# B&R Automation Studio project SuperTrak_Core
Automation Studio 4.7.4.67 SP; technology packages: mapp 5.11.1, mappView 5.11.2

## Configuration Simulation

CPU PC_any, AutomationRuntime B4.62, Build 4.1.2, Safety 0.0, Vc not defined

### Task classes (Cpu.sw)
```
Cyclic#1 (cycle 800 us, tolerance 0 us):
  ST_MainSim <- Source.ST_Core.ST_Main.prg
  ST_Logic <- Source.ST_Core.ST_Logic.prg
Cyclic#2 (cycle 800 us, tolerance 0 us):
  MainCtrl <- Source.Main.MainCtrl.prg
Cyclic#3 (cycle 50000 us):
  Alarms <- Source.Main.Alarms.prg
Cyclic#8 (cycle 800 us, tolerance 0 us):
  ST_Visu <- Source.ST_Core.ST_Visu.prg
DataObjects: Acp10sys, McAcpSys
Binaries: udbdef, mvLoader, TCData, arsvcreg, ashwac, arconfig, asfw, ashwd, iomap, User, Role, sysconf, Config_1, Config, Config_2, OpcUaMap, Acp10map, acp10cfg, McProfGen, McAcpSim, McAcpDrv, Config_3
Libraries: AsGuard, operator, runtime, astime, DevDetect, AsUDP, AsETH, AsIOTime, AsARCfg, AsIecCon, AsBrStr, AsIODiag, standard, ArEventLog, sys_lib, AsTCP, FileIO, brsystem, AsMem, DataObj, SuperTrak, AsArProf, StCom, CoTrace, AsZip, asstring, AsEthIP, AsPciStr, AsBrMath, MpAlarmX, MpBase, MpServer, MpCom, AsArLog, NcGlobal, aspciext, aruser, powerlnk
```

### Hardware
```
5LS182.6-2 : 5LS182.6-2 v1.3.1.0  [SL -> PC.SL4]
PC : PC_any v1.1.0.0 (OrderNumber=PC)
  Connector IF3:
    InaPort = 11159
  ConfigurationID = SuperTrak_Core_Simulation
  VolatileGlobalPvSize = 131070
  SystemTick = 400
  TaskClassIdleTime = 400
  Cyclic1Duration = 800
  Cyclic1Tolerance = 0
  Cyclic1Stack = 65535
  Cyclic1Output = 1
  Cyclic2Duration = 800
  Cyclic2Tolerance = 0
  Cyclic2Stack = 65535
  Cyclic3Duration = 50000
  Cyclic8Duration = 800
  Cyclic8Tolerance = 0
  FileDevice1
  FileDeviceName1 = USER
  FileDevicePath1 = ../../../../Logical/ConfigFiles
  FtpUser1
  FtpUsername1 = br
  FtpUserPassword1 = QMhL/dtrmhlR40mhXiUTZRHGDCdjSPoAwBd7aMiCRQw=
  FtpUserSalt1 = /GvO8l4J
  FTPAccessRight1 = 0
  WebServerWebDir = C:\web\
  ActivateOpcUa = 1
  OpcUaInformationModels_PV_Version = 1
```

## Configuration Standard_PC_TS77_04

CPU 5PC900.TS77-04, AutomationRuntime C4.72, Build 4.1.2, Safety 1.10, Vc V4.33.0

### Task classes (Cpu.sw)
```
Cyclic#1 (cycle 800 us, tolerance 0 us):
  ST_Main <- Source.ST_Core.ST_Main.prg
  ST_Logic <- Source.ST_Core.ST_Logic.prg
Cyclic#2 (cycle 800 us, tolerance 0 us):
  MainCtrl <- Source.Main.MainCtrl.prg
Cyclic#3:
  Alarms <- Source.Main.Alarms.prg
Cyclic#4:
  ST_Visu <- Source.ST_Core.ST_Visu.prg
Binaries: udbdef, mvLoader, TCData, arsvcreg, arconfig, User, Config, ashwd, Config_1, sysconf, ashwac, Role, asfw, iomap
Libraries: AsBrMath, AsGuard, operator, runtime, astime, DevDetect, AsUDP, AsETH, AsIOTime, AsARCfg, AsIecCon, AsBrStr, AsIODiag, standard, ArEventLog, sys_lib, AsTCP, FileIO, brsystem, AsMem, DataObj, SuperTrak, AsArProf, StCom, AsZip, asstring, AsEthIP, AsPciStr, MpBase, CoTrace, aruser, AsArLog, McBase, MpCom, MpAlarmX, MpServer, AsIOAcc
```

### Hardware
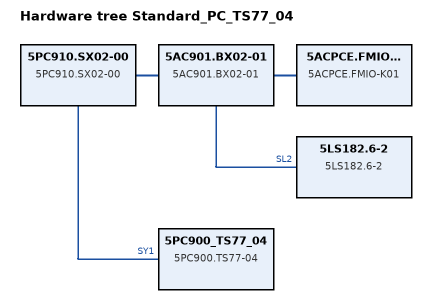
```
5AC901.BX02-01 : 5AC901.BX02-01 v1.1.1.0  [SY -> 5PC910.SX02-00.SY3]
5ACPCE.FMIO-K01 : 5ACPCE.FMIO-K01 v1.0.6.0  [SL -> 5AC901.BX02-01.SL1]
5LS182.6-2 : 5LS182.6-2 v1.4.0.0  [SL -> 5AC901.BX02-01.SL2]
  Connector IF1:
    CycleTime = 400
5PC900_TS77_04 : 5PC900.TS77-04 v2.0.1.0  [SY -> 5PC910.SX02-00.SY1]
  ConfigurationID = SuperTrak_Core_Standard_PC_TS77_04
  UserPartitionSize = 200
  RemMemDevice = PCI.2.LS182.SRAM
  RemMemSize = 500
  SystemTick = 400
  TaskClassIdleTime = 400
  Cyclic1Duration = 800
  Cyclic1Tolerance = 0
  Cyclic1Output = 1
  Cyclic2Duration = 800
  Cyclic2Tolerance = 0
  FileDevice1
  FileDeviceName1 = USER
  FileDevicePath1 = F:\SuperTrakCore
  EthernetDefaultGateway = 10.1.60.1
  ActivateDns = 1
  DnsDefaultDomain = br-automation.com
  DnsServer1 = 10.1.10.30
  FtpUser1
  FtpUsername1 = br
  FtpUserPassword1 = WcK/x6vgpRURITa0IoUtKo9v6R/fBL8dK5K21ruWyPI=
  FtpUserSalt1 = AV6KF4Bt
  FTPAccessRight1 = 0
  ActivateOpcUa = 1
  OpcUaInformationModels_PV_Version = 1
5PC910.SX02-00 : 5PC910.SX02-00 v2.0.2.0
  Connector IF1:
    AssignedOperatingSystem = ARemb
  Connector IF3:
    AssignedOperatingSystem = ARemb
    ActivateDevice = 1
    Mode = Manual
    InternetAddress = 10.1.60.55
    SubnetMask = 255.255.255.0
  Connector IF4:
    AssignedOperatingSystem = ARemb
    ActivateDevice = 1
    Mode = Manual
    InternetAddress = 10.11.10.12
    SubnetMask = 255.255.255.0
  Connector IF5:
    AssignedOperatingSystem = ARemb
  Connector IF6:
    AssignedOperatingSystem = ARemb
  Connector IF7:
    AssignedOperatingSystem = ARemb
  Connector IF8:
    AssignedOperatingSystem = ARemb
  Connector IF9:
    AssignedOperatingSystem = ARemb
```

## Configuration Standard_PC_TS77_1

CPU 5PC900.TS77-04, AutomationRuntime B4.45, Build 4.1.2, Vc V4.33.0, Safety 1.10

### Task classes (Cpu.sw)
```
Cyclic#1 (cycle 800 us, tolerance 0 us):
  ST_Main <- Source.ST_Core.ST_Main.prg
  ST_Logic <- Source.ST_Core.ST_Logic.prg
Cyclic#2 (cycle 800 us, tolerance 0 us):
  MainCtrl <- Source.Main.MainCtrl.prg
Cyclic#3:
  Alarms <- Source.Main.Alarms.prg
Cyclic#4:
  ST_Visu <- Source.ST_Core.ST_Visu.prg
Binaries: udbdef, mvLoader, TCData, arsvcreg, arconfig, User, Config, ashwd, Config_1, sysconf, ashwac, Role, asfw, iomap
Libraries: AsBrMath, AsGuard, operator, runtime, astime, DevDetect, AsUDP, AsETH, AsIOTime, AsARCfg, AsIecCon, AsBrStr, AsIODiag, standard, ArEventLog, sys_lib, AsTCP, FileIO, brsystem, AsMem, DataObj, SuperTrak, AsArProf, StCom, AsZip, asstring, AsEthIP, AsPciStr, MpBase, CoTrace, aruser, AsArLog, McBase, MpCom, MpAlarmX, MpServer
```

### Hardware
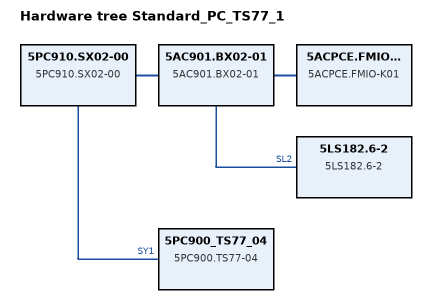
```
5AC901.BX02-01 : 5AC901.BX02-01 v1.1.1.0  [SY -> 5PC910.SX02-00.SY3]
5ACPCE.FMIO-K01 : 5ACPCE.FMIO-K01 v1.0.6.0  [SL -> 5AC901.BX02-01.SL1]
5LS182.6-2 : 5LS182.6-2 v1.3.1.0  [SL -> 5AC901.BX02-01.SL2]
  Connector IF1:
    CycleTime = 400
5PC900_TS77_04 : 5PC900.TS77-04 v2.0.0.0  [SY -> 5PC910.SX02-00.SY1]
  ConfigurationID = SuperTrak_Core_Standard_PC_TS77_04
  UserPartitionSize = 200
  RemMemDevice = PCI.2.LS182.SRAM
  RemMemSize = 500
  SystemTick = 400
  TaskClassIdleTime = 400
  Cyclic1Duration = 800
  Cyclic1Tolerance = 0
  Cyclic1Output = 1
  Cyclic2Duration = 800
  Cyclic2Tolerance = 0
  FileDevice1
  FileDeviceName1 = USER
  FileDevicePath1 = F:\SuperTrakCore
  FtpUser1
  FtpUsername1 = br
  FtpUserPassword1 = WcK/x6vgpRURITa0IoUtKo9v6R/fBL8dK5K21ruWyPI=
  FtpUserSalt1 = AV6KF4Bt
  FTPAccessRight1 = 0
  ActivateOpcUa = 1
  OpcUaInformationModels_PV_Version = 1
5PC910.SX02-00 : 5PC910.SX02-00 v2.0.1.0
  Connector IF1:
    AssignedOperatingSystem = ARemb
  Connector IF3:
    AssignedOperatingSystem = ARemb
    ActivateDevice = 1
    Mode = Manual
    InternetAddress = 10.11.10.50
    SubnetMask = 255.255.255.0
  Connector IF4:
    ActivateDevice = 1
    Mode = Manual
    InternetAddress = 10.1.10.11
    SubnetMask = 255.255.255.0
  Connector IF5:
    AssignedOperatingSystem = ARemb
  Connector IF6:
    AssignedOperatingSystem = ARemb
  Connector IF7:
    AssignedOperatingSystem = ARemb
  Connector IF8:
    AssignedOperatingSystem = ARemb
  Connector IF9:
    AssignedOperatingSystem = ARemb
```

### Config.mpalarmxcore - 5PC900_TS77_04/mappServices/Config.mpalarmxcore
```
Element gAlarmXCore (Type=mpalarmxcore)
  mapp.AlarmX.Core:
    Mapping:
      [0]:
        Alarm = 1
        [0]
  mapp.AlarmX.Core.Configuration:
    [0]:
      Name = Fault_0
      Message = {&ReportingSections}: Motor supply voltage out of range
      Behavior = UserDefined
        ReactionUntilAcknowledged = FALSE
        Recording:
          ActiveToInactive = FALSE
    [1]:
      Name = Fault_4
      Message = {&ReportingSections}: Excessive coil current
      Code = 4
      Behavior = UserDefined
        ReactionUntilAcknowledged = FALSE
        Recording:
          ActiveToInactive = FALSE
    [2]:
      Name = Fault_5
      Message = {&ReportingSections}: High temperature
      Code = 5
      Behavior = UserDefined
        ReactionUntilAcknowledged = FALSE
        Recording:
          ActiveToInactive = FALSE
    [3]:
      Name = Fault_7
      Message = {&ReportingSections}: Gateway network error
      Code = 7
      Behavior = UserDefined
        ReactionUntilAcknowledged = FALSE
        Recording:
          ActiveToInactive = FALSE
    [4]:
      Name = Fault_8
      Message = {&ReportingSections}: Excessive coil current (I2T)
      Code = 8
      Behavior = UserDefined
        ReactionUntilAcknowledged = FALSE
        Recording:
          ActiveToInactive = FALSE
    [5]:
      Name = Fault_9
      Message = {&ReportingSections}: Coil(s) unresponsive; check connection
      Code = 9
      Behavior = UserDefined
        ReactionUntilAcknowledged = FALSE
        Recording:
          ActiveToInactive = FALSE
    [6]:
      Name = Fault_11
      Message = {&ReportingSections}: Coil driver(s) shut down
      Code = 11
      Behavior = UserDefined
        ReactionUntilAcknowledged = FALSE
        Recording:
          ActiveToInactive = FALSE
    [7]:
      Name = Fault_14
      Message = {&ReportingSections}: Encoder calibration required
      Code = 14
      Behavior = UserDefined
        ReactionUntilAcknowledged = FALSE
        Recording:
          ActiveToInactive = FALSE
    [8]:
      Name = Fault_15
      Message = {&ReportingSections}: Excessive pallet following error
      Code = 15
      Behavior = UserDefined
        ReactionUntilAcknowledged = FALSE
        Recording:
          ActiveToInactive = FALSE
    [9]:
      Name = Fault_16
      Message = {&ReportingSections}: Unrecognized pallet(s) detected
      Code = 16
      Behavior = UserDefined
        ReactionUntilAcknowledged = FALSE
        Recording:
          ActiveToInactive = FALSE
    [10]:
      Name = Fault_19
      Message = {&ReportingSections}: Two pallets in collision deadlock
      Code = 19
      Behavior = UserDefined
        ReactionUntilAcknowledged = FALSE
        Recording:
          ActiveToInactive = FALSE
    [11]:
      Name = Fault_20
      Message = {&ReportingSections}: Pallet lost position feedback
      Code = 20
      Behavior = UserDefined
        ReactionUntilAcknowledged = FALSE
        Recording:
          ActiveToInactive = FALSE
    [12]:
      Name = Fault_21
      Message = {&ReportingSections}: Encoder read error
      Code = 21
      Behavior = UserDefined
        ReactionUntilAcknowledged = FALSE
        Recording:
          ActiveToInactive = FALSE
    [13]:
      Name = Fault_22
      Message = {&ReportingSections}: Coil driver error
      Code = 22
      Behavior = UserDefined
        ReactionUntilAcknowledged = FALSE
        Recording:
          ActiveToInactive = FALSE
    [14]:
      Name = Fault_23
      Message = {&ReportingSections}: Conflicting pallets detected
      Code = 23
      Behavior = UserDefined
        ReactionUntilAcknowledged = FALSE
        Recording:
          ActiveToInactive = FALSE
    [15]:
      Name = Fault_24
      Message = {&ReportingSections}: PLC interface heartbeat timeout
      Code = 24
      Behavior = UserDefined
        ReactionUntilAcknowledged = FALSE
        Recording:
          ActiveToInactive = FALSE
    [16]:
      Name = Fault_25
      Message = {&ReportingSections}: Encoder communication error
      Code = 25
      Behavior = UserDefined
        ReactionUntilAcknowledged = FALSE
        Recording:
          ActiveToInactive = FALSE
    [17]:
      Name = Fault_26
      Message = {&ReportingSections}: Disabled pallet arrived
      Code = 26
      Behavior = UserDefined
        ReactionUntilAcknowledged = FALSE
        Recording:
          ActiveToInactive = FALSE
    [18]:
      Name = Fault_27
      Message = {&ReportingSections}: Abnormal condition detected
      Code = 27
      Behavior = UserDefined
        ReactionUntilAcknowledged = FALSE
        Recording:
          ActiveToInactive = FALSE
    [19]:
      Name = Fault_28
      Message = {&ReportingSections}: Section disabled through configuration software
      Code = 28
      Behavior = UserDefined
        ReactionUntilAcknowledged = FALSE
        Recording:
          ActiveToInactive = FALSE
    [20]:
      Name = Fault_30
      Message = {&ReportingSections}: Hardware initialization error
      Code = 30
      Behavior = UserDefined
        ReactionUntilAcknowledged = FALSE
        Recording:
          ActiveToInactive = FALSE
    [21]:
      Name = Fault_31
      Message = Fatal abnormal condition detected
      Code = 31
      Behavior = UserDefined
        ReactionUntilAcknowledged = FALSE
        Recording:
          ActiveToInactive = FALSE
    [22]:
      Name = Warning_1
      Message = {&ReportingSections}: Application Warning
      Code = 1
      Behavior = UserDefined
    [23]:
      Name = Warning_4
      Message = {&ReportingSections}: Thermal sensor malfunction
      Code = 4
      Behavior = UserDefined
    [24]:
      Name = Warning_5
      Message = {&ReportingSections}: High temperature
      Code = 5
      Behavior = UserDefined
    [25]:
      Name = Warning_7
      Message = {&ReportingSections}: Gateway network warning
      Code = 7
      Behavior = UserDefined
    [26]:
      Name = Warning_8
      Message = {&ReportingSections}: Excessive coil current (I2T)
      Code = 8
      Behavior = UserDefined
    [27]:
      Name = Warning_9
      Message = {&ReportingSections}: Coil(s) unresponsive; check connection
      Code = 9
      Behavior = UserDefined
    [28]:
      Name = Warning_11
      Message = {&ReportingSections}: Pallet position correction was required
      Code = 11
      Behavior = UserDefined
    [29]:
      Name = Warning_12
      Message = {&ReportingSections}: Pallet ID tag warning
      Code = 12
      Behavior = UserDefined
    [30]:
      Name = Warning_13
      Message = {&ReportingSections}: Duplicate Pallet ID
      Code = 13
      Behavior = UserDefined
    [31]:
      Name = Warning_15
      Message = {&ReportingSections}: Counts out of range during encoder handoff
      Code = 15
      Behavior = UserDefined
    [32]:
      Name = Warning_16
      Message = {&ReportingSections}: Consecutive encoder readings out of range
      Code = 16
      Behavior = UserDefined
    [33]:
      Name = Warning_17
      Message = {&ReportingSections}: Invalid region configuration
      Code = 17
      Behavior = UserDefined
    [34]:
      Name = Warning_18
      Message = {&ReportingSections}: Invalid parameter configuration
      Code = 18
      Behavior = UserDefined
    [35]:
      Name = Warning_19
      Message = {&ReportingSections}: Command failed
      Code = 19
      Behavior = UserDefined
    [36]:
      Name = Warning_20
      Message = {&ReportingSections}: Invalid sync zone configuration
      Code = 20
      Behavior = UserDefined
    [37]:
      Name = Warning_21
      Message = {&ReportingSections}: Encoder read warning
      Code = 21
      Behavior = UserDefined
    [38]:
      Name = Warning_22
      Message = {&ReportingSections}: Coil driver warning
      Code = 22
      Behavior = UserDefined
    [39]:
      Name = Warning_23
      Message = {&ReportingSections}: Parameter save required
      Code = 23
      Behavior = UserDefined
    [40]:
      Name = Warning_24
      Message = {&ReportingSections}: Pallet destination updated
      Code = 24
      Behavior = UserDefined
    [41]:
      Name = Warning_25
      Message = {&ReportingSections}: Encoder communication warning
      Code = 25
      Behavior = UserDefined
    [42]:
      Name = Warning_26
      Message = {&ReportingSections}: Disabled pallet arrived
      Code = 26
      Behavior = UserDefined
    [43]:
      Name = Warning_27
      Message = {&ReportingSections}: Too many pallets
      Code = 27
      Behavior = UserDefined
    [44]:
      Name = Warning_29
      Message = {&ReportingSections}: Excessive pallet settling time
      Code = 29
      Behavior = UserDefined
    [45]:
      Name = Warning_30
      Message = {&ReportingSections}: Controller health warning
      Code = 30
      Behavior = UserDefined
    [46]:
      Name = Warning_31
      Message = Abnormal condition detected
      Code = 31
      Behavior = UserDefined
  mapp.AlarmX.Core.Snippets:
    [0]:
      Key = ReportingSections
      Value:
        PV = ::Alarms:reportingSections
```

### Config_1.mpalarmxhistory - 5PC900_TS77_04/mappServices/Config_1.mpalarmxhistory
```
Element gAlarmXHistory (Type=mpalarmxhistory)
  mapp.AlarmX.History:
    Memory:
      MemorySize = 2000
```

## Logical view

Binary libraries used (declarations not repeated): AsGuard, operator, runtime, astime, DevDetect 1.00.0, AsUDP, AsETH, AsIOTime, AsARCfg, AsIecCon, AsBrStr, AsIODiag, standard, ArEventLog, sys_lib, AsTCP, FileIO, brsystem, AsMem, SuperTrak 0.22.4, AsArProf, StCom 5.04.0, CoTrace 5.00.1, AsZip, DataObj, asstring, AsEthIP, AsPciStr, AsBrMath, AsArLog, NcGlobal 5.06.0, McBase 5.04.9, AsIOAcc, MpServer 5.11.0, MpAlarmX 5.11.1, MpBase, MpCom, StCom_OLD 5.03.0, SuperTrak_OLD 0.06.2

### Global.var - Global variables
```iecst
VAR
	gStLink : StLinkType; (*StCom library communication variable*)
	gStCyclicControlData : {REDUND_UNREPLICABLE} ARRAY[0..499] OF USINT := [500(0)]; (*Cyclic control buffer (to SuperTrak)*)
	gStCyclicStatusData : {REDUND_UNREPLICABLE} ARRAY[0..499] OF USINT := [500(0)]; (*Cyclic status buffer (from SuperTrak)*)
	gStServiceChannelReqData : {REDUND_UNREPLICABLE} ARRAY[0..127] OF USINT := [128(0)]; (*Service channel request buffer (to SuperTrak)*)
	gStServiceChannelResData : {REDUND_UNREPLICABLE} ARRAY[0..127] OF USINT := [128(0)]; (*Service channel response buffer (from SuperTrak)*)
END_VAR
VAR CONSTANT
	CONFIG_ST_MAX_SECTIONS : USINT := 4; (*Number of sections on the SuperTrak system*)
	CONFIG_ST_MAX_PALLETS : USINT := 40; (*Maximum number of pallets on the SuperTrak system*)
	CONFIG_ST_MAX_TARGETS : USINT := 40; (*Maximum number of targets on the SuperTrak system !!! MUST BE DIVISIBLE BY 4*)
	CONFIG_ST_MAX_COMMANDS : USINT := 24; (*Maximum number of commands, which should be executed in parallel on the SuperTrak system*)
END_VAR
VAR
	gSuperTrak : SysTrak_typ; (*Main control task for SuperTrak system*)
	testString : STRING[200];
END_VAR
```

### Global.typ - Global data types
```iecst
TYPE
	SysCmds_typ : 	STRUCT  (*System-wide commands to control SuperTrak*)
		Enable : BOOL; (*Commands sections to power on and locate pallets*)
		Start : BOOL; (*Begin application code & pallet routing*)
		ErrorReset : BOOL; (*Acknowledges recoverable & inactive errors*)
	END_STRUCT;
	SysPalletPar_typ : 	STRUCT  (*Configuration parameters for Pallet commands*)
		Config : SysReleaseConfig_typ; (*Includes motion parameters for specific pallet*)
		IncrementOffset : BOOL; (*Command to add a specific offset to the pallet at the target (e.g. for calibration) Relative*)
		ReleaseToOffset : BOOL; (*Command to add a specific offset to the pallet at the target (e.g. for calibration) Absolute*)
		ReleaseToTarget : BOOL; (*Command to release the pallet ID to a specified destination target*)
		Synchronize : BOOL;
	END_STRUCT;
	SysPalletStatus_typ : 	STRUCT  (*Status information for Pallets*)
		Section : USINT; (*Pallet current section*)
		Position : REAL; (*Pallet current position along section*)
		Velocity : REAL; (*Pallet current set velocity*)
		Acceleration : REAL; (*Pallet current set acceleration*)
		PalletReleased : BOOL; (*Pallet has been released. Used to acknowledge ReleaseToTarget command*)
		PalletAllocated : BOOL;
		DestinationTarget : UINT;
	END_STRUCT;
	SysPar_typ : 	STRUCT  (*Configuration parameters for System commands*)
		System : SysSystemPar_typ; (*System-wide parameters*)
		Pallet : ARRAY[0..CONFIG_ST_MAX_PALLETS]OF SysPalletPar_typ; (*Pallet-specific parameters*)
		Target : ARRAY[0..CONFIG_ST_MAX_TARGETS]OF SysTargetsPar_typ; (*Target-specific parameters*)
	END_STRUCT;
	SysReleaseConfig_typ : 	STRUCT  (*Release configuration type*)
		TargetOffset : REAL;
		Velocity : UINT; (*Set velocity for next movement [mm/s]*)
		Acceleration : UINT; (*Set acceleration for next movement [mm/s2]*)
		Direction : StParamAdvReleaseConfigDirEnum; (*Direction of movement (assumes facing an upright track). Can use constants: stCOM_DIR_RIGHT, stCOM_DIR_LEFT*)
		DestinationTarget : USINT; (*Destination target of an absolute movement*)
		IncrementOffset : REAL;
		SyncTarget : UDINT;
	END_STRUCT;
	SysSectionDetails_typ : 	STRUCT  (*Status information for specific section*)
		MotorTemp : ARRAY[0..5]OF REAL; (*Motor temperatures [C]. Each section has 10 temp sensors*)
		MotorVoltage : REAL; (*Motor voltage [V]*)
		ElectronicsTemp : REAL; (*Electronics temps [C]*)
	END_STRUCT;
	SysSectionDiag_typ : 	STRUCT  (*Diagnostic information for a section*)
		Enabled : BOOL; (*Section is enabled*)
		UnrecPallPresent : BOOL; (*Indicates whether pallets on the section are not recognized*)
		MotorPowerOn : BOOL; (*Indicates whether the motor power is on*)
		PalletsRecovering : BOOL; (*Indicates whether pallets are currently recovering*)
		LocatingPallets : BOOL; (*Indicates whether pallets are being automatically 'jogged' so that their location can be determined*)
		DisabledExternally : BOOL; (*Indicates if the section is disabled due to an external condition*)
		WarningActive : BOOL;
		FaultActive : BOOL;
		Warnings : ARRAY[0..31]OF BOOL; (*Warning bits for the section- used as alarm conditions*)
		Faults : ARRAY[0..31]OF BOOL; (*Fault bits for the section- usued as alarm conditions*)
	END_STRUCT;
	SysSectionStatus_typ : 	STRUCT  (*Status categories for sections*)
		Right : SysSectionDetails_typ; (*Right driver board*)
		Diag : SysSectionDiag_typ; (*Diagnostics information*)
		Left : SysSectionDetails_typ; (*Left driver board*)
		IsCurveSection : BOOL; (*Determines if the section is a curve or not*)
	END_STRUCT;
	SysStatus_typ : 	STRUCT  (*Status categories*)
		System : SysSystemStatus_typ; (*System-wide status*)
		Section : ARRAY[0..CONFIG_ST_MAX_SECTIONS]OF SysSectionStatus_typ; (*Individual section status*)
		Target : ARRAY[0..CONFIG_ST_MAX_TARGETS]OF SysTargetStatus_typ; (*Individual target status*)
		Pallet : ARRAY[0..CONFIG_ST_MAX_PALLETS]OF SysPalletStatus_typ; (*Individual pallet status*)
	END_STRUCT;
	SysSystemPar_typ : 	STRUCT  (*System-wide configuration parameters*)
		RecoveryTarget : USINT; (*Defines a target for pallets to recover to after a system halt*)
		RecoveryDirection : StParamAdvReleaseConfigDirEnum; (*Defines a direction for pallets to head towards the recovery target*)
		RecoveryAccel : UINT; (*Defines an acceleration parameter for pallets while moving towards a recovery target*)
		RecoveryVelocity : UINT; (*Defines a maximum velocity for pallets while moving towards a recovery target*)
	END_STRUCT;
	SysSystemStatus_typ : 	STRUCT  (*System-wide status information*)
		Enabled : BOOL; (*Indicates that all sections are powered*)
		Ready : BOOL; (*Indicates that sections are powered and shuttles have been located*)
		Running : BOOL; (*Indicates that the application code is active and shuttle routing is underway *)
		WarningActive : BOOL; (*Indicates that at least one system warning is active*)
		FaultsActive : BOOL; (*Indicates that at least one system fault is active*)
		Warnings : ARRAY[0..31]OF BOOL; (*Alarm status bits for system warnings*)
		Faults : ARRAY[0..31]OF BOOL; (*Alarm status bits for system faults*)
		ActiveSections : USINT;
		ActivePallets : USINT; (*Counts number of active pallets on the system*)
		EMA_Throughput : REAL := 0.0; (*Calculates Exponential Moving Average of the throughput*)
		Throughput : REAL; (*Calculates instantaneous system throughput*)
	END_STRUCT;
	SysTargetsPar_typ : 	STRUCT  (*Target configuration parameters*)
		Config : SysReleaseConfig_typ; (*Motion parameter configuration datatype*)
		IncrementOffset : BOOL; (*Command to add a specific offset to the pallet at the target (e.g. for calibration) Relative*)
		ReleaseToOffset : BOOL; (*Command to add a specific offset to the pallet at the target (e.g. for calibration) Absolute*)
		ReleaseToTarget : BOOL; (*Command to release the pallet at the target to a specified destination target*)
	END_STRUCT;
	SysTargetStatus_typ : 	STRUCT  (*Target status information. Used to detect pallet presence & ID*)
		PalletId : USINT; (*Pallet ID*)
		PalletReleased : BOOL; (*Pallet has been released. Used to acknowledge ReleaseToTarget command*)
		PalletPreArrival : BOOL; (*Pallet is about to arrive at the target*)
		PalletPresent : BOOL; (*Pallet is detected at the target*)
		Section : UINT; (*Configured Section for the target*)
		Position : REAL; (*Configured Position for the target [mm]*)
		PalletHovering : BOOL; (*Pallet is detected over (but not necessarily destined for) a target with Hover enabled*)
	END_STRUCT;
	SysTrak_typ : 	STRUCT  (*High level control structure for handling the SuperTrak system*)
		Cmds : SysCmds_typ; (*Commands datatype. INPUTS to the SuperTrak*)
		Par : SysPar_typ; (*Parameters datatype. INPUTS to the SuperTrak*)
		Status : SysStatus_typ; (*Status datatype. OUTPUTS from the SuperTrak*)
	END_STRUCT;
END_TYPE
```


### Package Logical/Source - Project source code

### Package Logical/Source/ST_Core - Core SuperTrak Functionality

### Program Logical/Source/ST_Core/ST_Main (IEC) - Manages ST service channel

#### Variables.var
```iecst
(********************************************************************
 * Copyright ATS Automation Tooling Systems, Inc. 2015
 * All rights reserved.
 ********************************************************************
 * Local variables
 ********************************************************************)
(*ServiceChannel Handling*)
VAR
	SuperTrakControlInterface : ARRAY[0..stMAX_CONTROL_IF_INDEX] OF SuperTrakControlInterface_t := [stMAX_CONTROL_IF_COUNT((0))];
	ServiceChannelData : ServiceChannel_t := (0);
	pResView : REFERENCE TO ServiceChannelHeader_t;
	pReqView : REFERENCE TO ServiceChannelHeader_t;
END_VAR
(*SuperTrak Init Parameters*)
VAR
	ARSimIPAddress : STRING[15] := '127.0.0.1'; (*IP Adress of the ArSim*)
	EthernetInterfaces : STRING[31] := 'IF3,IF4'; (*Existing Ethernet Interfaces on APC*)
	StoragePath : STRING[127];
END_VAR
(*Insert your comment here.*)
VAR
	i : UINT := 0;
	status : UINT := 0;
	count : UINT := 0;
	digitalInputFunction : ARRAY[0..7] OF UINT := [8(0)];
	udintValue : UDINT;
	uintValue : UINT;
	taskName : STRING[10];
	mvCounter : INT;
	IsSimulation : BOOL;
	SuperTrakStoragePath : STRING[80];
	taskGroup : USINT;
END_VAR
```

#### Main.st
```iecst
(*********************************************************************************
 * Copyright: ATS Automation Tooling Systems, Inc. 2015
 *     All rights reserved.
 *********************************************************************************
 *********************************************************************************
 * Description:
 * -------------------------------------------------------------------------------
 * This task configures the internal communication structure AND controlls
 * the SuperTrak system.
 *********************************************************************************)

PROGRAM _INIT
// SuperTrak initialization
(* DiagCpuIsSimulated() returns TRUE if "Activate Simulation" is enabled. *)
	IsSimulation := DiagCpuIsSimulated();

(* DiagCpuIsSimulated() returns FALSE if the project configuration specifies
 * ARsim. Assume simulation mode IF this task is named 'ST_MainSim'.
 *)
	taskName := '';
	status := ST_name(0, ADR(taskName), ADR(taskGroup));

	IF (taskName = 'ST_MainSim') THEN
		IsSimulation := TRUE;
	END_IF;

	IF (IsSimulation) THEN
		(* This path can be customized as needed *)
		SuperTrakStoragePath := '/DEVICE=../../../../Logical/ConfigFiles';
		//SuperTrakStoragePath	:= '/DEVICE=C:\SuperTrakCfg\SuperTrakCore';
	ELSE
		(* CFast card USER partition *)
		SuperTrakStoragePath := '/DEVICE=F:\SuperTrakCore';
	END_IF;

	// SuperTrak Init function call
	SuperTrakInit(SuperTrakStoragePath, ARSimIPAddress, EthernetInterfaces);

	// Service Channel initialization
	ServiceChannelData.channelId    		:= 1;
	ServiceChannelData.pRequestHeader		:= ADR(gStServiceChannelReqData);
	ServiceChannelData.pResponseHeader		:= ADR(gStServiceChannelResData);
	ServiceChannelData.pRequestValues     	:= ADR(gStServiceChannelReqData) + SIZEOF(ServiceChannelHeader_t);
	ServiceChannelData.pResponseValues    	:= ADR(gStServiceChannelResData) + SIZEOF(ServiceChannelHeader_t);
	ServiceChannelData.requestBufferSize  	:= SIZEOF(gStServiceChannelReqData);
	ServiceChannelData.responseBufferSize  	:= SIZEOF(gStServiceChannelResData);
	ServiceChannelData.state     			:= scSTATE_RECV;

	pResView ACCESS ADR(gStServiceChannelResData);
	pReqView ACCESS ADR(gStServiceChannelReqData);

	// Command interface mapping
	SuperTrakControlInterface[0].pControl  	:= ADR(gStCyclicControlData);
	SuperTrakControlInterface[0].pStatus   	:= ADR(gStCyclicStatusData);
	SuperTrakControlInterface[0].controlSize:= SIZEOF(gStCyclicControlData);
	SuperTrakControlInterface[0].statusSize := SIZEOF(gStCyclicStatusData);

	(* De-configure any "Allow Section Enable" inputs *)
	(* Parameter 1092: Parameter Array Length (UDINT) *)
	(* Parameter 1200: Digital Input Function (UINT) *)
	status := SuperTrakServChanRead(0, 1092, 1200 - 1024, 1, ADR(udintValue), SIZEOF(udintValue));

	IF (status = scERR_SUCCESS) THEN
		count := MIN(UDINT_TO_UINT(udintValue),
		SIZEOF(digitalInputFunction) / SIZEOF(digitalInputFunction[0]));

		status := SuperTrakServChanRead(0, 1200, 0, count, ADR(digitalInputFunction), SIZEOF(digitalInputFunction));

		IF (status = scERR_SUCCESS) THEN
			FOR i := 0 TO count - 1 DO
				(* Input Function 25: Allow Section Enable *)
				IF (digitalInputFunction[i] = 25) THEN
					(* Input Function 0: Not Configured *)
					digitalInputFunction[i] := 0;
					status := SuperTrakServChanWrite(0, 1200, i, 1, ADR(digitalInputFunction[i]), SIZEOF(digitalInputFunction[i]));
				END_IF;
			END_FOR;
		END_IF;
	END_IF;

	(* Ensure that control interface revision 0 is selected *)
	(* Parameter 1444: Control Interface Revision (UINT) *)
	status := SuperTrakServChanRead(0, 1444, 0, 1, ADR(uintValue), SIZEOF(uintValue));

	IF (status = scERR_SUCCESS) THEN
		IF (uintValue <> 0) THEN
			uintValue := 0;
			status := SuperTrakServChanWrite(0, 1444, 0, 1, ADR(uintValue), SIZEOF(uintValue));
		END_IF;
	END_IF;

END_PROGRAM

PROGRAM _CYCLIC

	mvCounter	:= mvCounter + 1;

	// Cylcic SuperTrak control
	SuperTrakCyclic1();

	// Map internal communication structure
	FOR i := 0 TO stMAX_CONTROL_IF_INDEX DO
		SuperTrakProcessControl(i, SuperTrakControlInterface[i]);
	END_FOR;

	// Service channel handling
	IF ServiceChannelData.state = scSTATE_RECV AND
		pReqView.sequence <> pResView.sequence THEN
		ServiceChannelData.requestSequence  := pReqView.sequence;
		ServiceChannelData.state    		:= scSTATE_EXEC;
	ELSIF ServiceChannelData.state = scSTATE_EXEC OR ServiceChannelData.state = scSTATE_WAIT THEN
		SuperTrakServiceChannel(ServiceChannelData);
	ELSIF ServiceChannelData.state = scSTATE_SEND THEN
		ServiceChannelData.state    		:= scSTATE_RECV;
	END_IF;

END_PROGRAM

PROGRAM _EXIT

 // Clear internal memory
	SuperTrakExit();

END_PROGRAM
```

### Program Logical/Source/ST_Core/ST_Logic (IEC, version 1.00.0) - Accepts commands from gSuperTrak. Manages System, Section, and Pallet function blocks

#### Main.st - Cyclic code
```iecst
(*********************************************************************************
 * Copyright: Bernecker + Rainer
 * Author:  Bernecker + Rainer
 * Created:  July 27, 2016/10:44 AM
 *********************************************************************************
 *********************************************************************************
 * Version History:
 * -------------------------------------------------------------------------------
 * V 1.00.0   July 27, 2016/10:44 AM  First Version
 * V 1.10.0	  January 3, 2018/4:30 PM	Updated to work with new gSuperTrak
										command structure
 *********************************************************************************
 * Description:

	This task accepts commands and parameters from the gSuperTrak control structure,
	and writes new status information to the same structure. ST_Logic should not
	be necessary to modify, and can be used as a starting point for applications.
 *********************************************************************************)

PROGRAM _INIT

 (*************************************************************************************************)
 (*************************************************************************************************)
 (* FUNCTION BLOCK CONFIGURATION *)

 // Configure the internal communication structure to/from SuperTrak
	SuperTrakControlParameters.NrOfCommands        	:= CONFIG_ST_MAX_COMMANDS;
	SuperTrakControlParameters.NrOfPallets        	:= CONFIG_ST_MAX_PALLETS;
	SuperTrakControlParameters.NrOfSections        	:= CONFIG_ST_MAX_SECTIONS;
	SuperTrakControlParameters.NrOfTargets        	:= CONFIG_ST_MAX_TARGETS;

	(*************************************************************************************************)
	(*************************************************************************************************)
	(* FUNCTION BLOCK INITIALIZATION *)

	// Initialize the function block, handling the communication to/from SuperTrak
	StControl_0.StLink       				:= ADR(gStLink);
	StControl_0.Enable       				:= TRUE;
	StControl_0.Parameters      			:= ADR(SuperTrakControlParameters);
	StControl_0.StCtrlData      			:= ADR(gStCyclicControlData);
	StControl_0.StCtrlDataSize     			:= SIZEOF(gStCyclicControlData);
	StControl_0.StStatData      			:= ADR(gStCyclicStatusData);
	StControl_0.StStatDataSize     			:= SIZEOF(gStCyclicStatusData);
	StControl_0.StServChRequestData   		:= ADR(gStServiceChannelReqData);
	StControl_0.StServChRequestDataSize  	:= SIZEOF(gStServiceChannelReqData);
	StControl_0.StServChResponseData  		:= ADR(gStServiceChannelResData);
	StControl_0.StServChResponseDataSize 	:= SIZEOF(gStServiceChannelResData);

	// Initialize parameter read function block to pull status information from SuperTrak
	StReadPnu_0.StLink						:= ADR(gStLink);
	StReadPnu_0.Parameters					:= ADR(ReadPnuPara[0]);
	StReadPnu_0.DataAddress					:= ADR(ReadDataBuffer[0].Entry);
	StReadPnu_0.DataSize					:= SIZEOF(ReadDataBuffer[0].Entry);

	// Initialize parameter write function block to push parameter information to the SuperTrak
	StWritePnu_0.StLink						:= ADR(gStLink);
	StWritePnu_0.Parameters					:= ADR(WritePnuPara[0]);
	StWritePnu_0.DataAddress				:= ADR(WriteDataBuffer[0].Entry);
	StWritePnu_0.DataSize					:= SIZEOF(WriteDataBuffer[0].Entry);

	// Initialize parameter inputs to Section control function block
	FOR Index := 0 TO (SIZEOF(StSection_) / SIZEOF(StSection_[0])) - 1 DO
		SuperTrakSectionParameters[Index].Reserved;
	END_FOR;

	// Initialize parameter inputs to Target control function block
	FOR Index := 0 TO (SIZEOF(StTargetExt_) / SIZEOF(StTargetExt_[0])) - 1 DO
		SuperTrakTargetParameters[Index].AdvancedReleaseConfig.DestinationTarget	:= 15;
		SuperTrakTargetParameters[Index].AdvancedReleaseConfig.Direction			:= stCOM_DIR_RIGHT;
		SuperTrakTargetParameters[Index].PalletConfig.Motion.Acceleration			:= 500;//mm/s^2
		SuperTrakTargetParameters[Index].PalletConfig.Motion.Velocity				:= 1000;//mm/s
	END_FOR;

	// Initialize parameter inputs to Pallet control function blocks
	FOR Index := 0 TO (SIZEOF(StPallet_) / SIZEOF(StPallet_[0])) - 1 DO
		SuperTrakPalletParameters[Index].AdvancedReleaseConfig.DestinationTarget	:= 15;
		SuperTrakPalletParameters[Index].AdvancedReleaseConfig.Direction			:= stCOM_DIR_RIGHT;
		SuperTrakPalletParameters[Index].PalletConfig.Motion.Acceleration			:= 500;//mm/s^2
		SuperTrakPalletParameters[Index].PalletConfig.Motion.Velocity				:= 1000;//mm/s
	END_FOR;

	// Initialize the function blocks, controlling a single section
	FOR Index := 0 TO (SIZEOF(StSection_) / SIZEOF(StSection_[0])) - 1 DO
		StSection_[Index].StLink    		:= ADR(gStLink);
		StSection_[Index].Parameters  		:= ADR(SuperTrakSectionParameters[Index]);
		StSection_[Index].Section   		:= Index;
	END_FOR;

	// Initialize the function blocks, controlling a single target
	FOR Index := 0 TO (SIZEOF(StTargetExt_) / SIZEOF(StTargetExt_[0])) - 1 DO
		StTargetExt_[Index].StLink    		:= ADR(gStLink);
		StTargetExt_[Index].Parameters   	:= ADR(SuperTrakTargetParameters[Index]);
		StTargetExt_[Index].Target    		:= Index;
	END_FOR;

	// Initialize the function blocks controlling a single pallet
	FOR Index := 0 TO (SIZEOF(StPallet_) / SIZEOF(StPallet_[0])) - 1 DO
		StPallet_[Index].StLink				:= ADR(gStLink);
		StPallet_[Index].Parameters			:= ADR(SuperTrakPalletParameters[Index]);
		StPallet_[Index].PalletID			:= Index;
	END_FOR;

END_PROGRAM

PROGRAM _CYCLIC

 (*************************************************************************************************)
 (*************************************************************************************************)
 (* FUNCTION BLOCK ENABLE *)

 // Wait for StControl to be active, before enalbing all other function blocks
	IF StControl_0.Active THEN
		// Loop thru all StSection function blocks
		FOR Index := 0 TO (SIZEOF(StSection_) / SIZEOF(StSection_[0])) - 1 DO
			// Enable StSection
			StSection_[Index].Enable     := TRUE;
		END_FOR;

		// Loop thru all StTargetExt function blocks
		FOR Index := 0 TO (SIZEOF(StTargetExt_) / SIZEOF(StTargetExt_[0])) - 1 DO
			// Enable StTargetExt
			StTargetExt_[Index].Enable     := TRUE;
		END_FOR;

		// Loop thru all StPallet function blocks
		FOR Index := 0 TO (SIZEOF(StPallet_) /SIZEOF(StPallet_[0]) - 1) DO
			// Enable StPallet
			StPallet_[Index].Enable			:= TRUE;
		END_FOR;

	END_IF;

	(*************************************************************************************************)
	(*************************************************************************************************)
	(* ENABLE / DISABLE SUPERTRAK SECTIONS *)

	// Wait for command, to enable all sections
	IF gSuperTrak.Cmds.Enable THEN
		// Loop thru all StSection function blocks
		FOR Index := 0 TO (SIZEOF(StSection_) / SIZEOF(StSection_[0])) - 1 DO
			// Check if section is ready to be enalbed
			IF StSection_[Index].MotorPowerOn AND NOT StSection_[Index].Error THEN
				// Enable section
				StSection_[Index].EnableSection   := TRUE;
			END_IF;
		END_FOR;

		// If command is reset, disable all sections
	ELSE
		// Loop thru all StSection function blocks
		FOR Index := 0 TO (SIZEOF(StSection_) / SIZEOF(StSection_[0])) - 1 DO
			// Disable section
			StSection_[Index].EnableSection		:= FALSE;
			//StSection_[Index].Enable			:= FALSE;
		END_FOR;
	END_IF;

	(*************************************************************************************************)
	(*************************************************************************************************)
	(* PALLET ROUTING AROUND THE SYSTEM - ACCEPT INPUTS FROM gSUPERTRAK *)

	// Check if all sections are enabled, before setting any commands
	IF StControl_0.SectionsEnabled THEN

		// Set the system status bit POWERED high
		gSuperTrak.Status.System.Enabled		:= TRUE;

		// Loop through all possible targets to accept new configuration parameters & release commands
		FOR Index := 1 TO ((SIZEOF(StTargetExt_) / SIZEOF(StTargetExt_[0]))-1) DO
			CASE StTargetState[Index] OF
				0:	// Begin state machine if a release command is sent by the main application
					IF gSuperTrak.Status.Target[Index].PalletPresent AND
						(gSuperTrak.Par.Target[Index].ReleaseToTarget OR
						gSuperTrak.Par.Target[Index].ReleaseToOffset OR
						gSuperTrak.Par.Target[Index].IncrementOffset) THEN

						// Grab all command information within the same cycle, in case MainCtrl modifies these commands in subsequent cycles
						IF gSuperTrak.Par.Target[Index].ReleaseToTarget THEN
							releaseModeTarget[Index]				:= 0;
						ELSIF gSuperTrak.Par.Target[Index].ReleaseToOffset THEN
							releaseModeTarget[Index]				:= 1;
						ELSIF gSuperTrak.Par.Target[Index].IncrementOffset THEN
							releaseModeTarget[Index]				:= 2;
						END_IF;

						// Do the same for motion parameters & release config
						SuperTrakTargetParameters[Index].PalletConfig.Motion.Acceleration			:= gSuperTrak.Par.Target[Index].Config.Acceleration;
						SuperTrakTargetParameters[Index].PalletConfig.Motion.Velocity				:= gSuperTrak.Par.Target[Index].Config.Velocity;
						SuperTrakTargetParameters[Index].AdvancedReleaseConfig.DestinationTarget	:= gSuperTrak.Par.Target[Index].Config.DestinationTarget;
						SuperTrakTargetParameters[Index].AdvancedReleaseConfig.TargetOffset			:= gSuperTrak.Par.Target[Index].Config.TargetOffset;
						SuperTrakTargetParameters[Index].AdvancedReleaseConfig.IncrementalOffset	:= gSuperTrak.Par.Target[Index].Config.IncrementOffset;
						SuperTrakTargetParameters[Index].AdvancedReleaseConfig.Direction			:= gSuperTrak.Par.Target[Index].Config.Direction;

						StTargetState[Index]	:= 1;
					END_IF;
				1:	// Update motion parameters for the commanded movement
					StTargetExt_[Index].SetPalletMotionPar										:= TRUE;

					// Once the update is complete, move to the next state in the state machine
					IF StTargetExt_[Index].CommandDone THEN
						StTargetExt_[Index].SetPalletMotionPar									:= FALSE;
						StTargetState[Index]													:= 2;
					END_IF;

				2:	// Update destination target and travel direction for the commanded movement
					StTargetExt_[Index].Update													:= TRUE;

					// Once the update is complete, move to the next state in the state machine
					IF StTargetExt_[Index].UpdateDone THEN
						StTargetExt_[Index].Update												:= FALSE;
						StTargetState[Index]													:= 3;
					END_IF;
				3:
					//Pass the release command (either target or offset) to the StTarget function block and execute
					CASE releaseModeTarget[Index] OF
						0:		StTargetExt_[Index].ReleaseToTarget								:= TRUE;
						1:		StTargetExt_[Index].ReleaseToOffset								:= TRUE;
						2:		StTargetExt_[Index].IncrementOffset								:= TRUE;
					END_CASE;

					IF StTargetExt_[Index].CommandDone THEN
						StTargetExt_[Index].ReleaseToTarget										:= FALSE;
						StTargetExt_[Index].ReleaseToOffset										:= FALSE;
						StTargetExt_[Index].IncrementOffset										:= FALSE;
						StTargetState[Index]													:= 4;
					END_IF;
				4:
					// Once the pallet is released, notify the main application w/ PalletReleased and reset the state machine
					gSuperTrak.Status.Target[Index].PalletReleased								:= TRUE;
					IF gSuperTrak.Par.Target[Index].ReleaseToTarget = FALSE AND gSuperTrak.Par.Target[Index].ReleaseToOffset = FALSE AND gSuperTrak.Par.Target[Index].IncrementOffset = FALSE THEN
						gSuperTrak.Status.Target[Index].PalletReleased							:= FALSE;
						StTargetState[Index]													:= 0;
					END_IF;

				5:
				6:
				7:
				8:
				9:

			END_CASE;
		END_FOR;

		// Loop through all possible pallets to accept new configuration parameters & release commands
		FOR Index := 0 TO ((SIZEOF(StPallet_) / SIZEOF(StPallet_[0]))-1) DO
			CASE StPalletState[Index] OF
				0:	// Begin state machine if a release command is sent by the main application
					IF gSuperTrak.Par.Pallet[Index].ReleaseToTarget OR
						gSuperTrak.Par.Pallet[Index].ReleaseToOffset OR
						gSuperTrak.Par.Pallet[Index].IncrementOffset THEN

						// Grab all command information within the same cycle, in case MainCtrl modifies these commands in subsequent cycles
						IF gSuperTrak.Par.Pallet[Index].ReleaseToTarget THEN
							releaseModePallet[Index]			:= 0;
						ELSIF gSuperTrak.Par.Pallet[Index].ReleaseToOffset THEN
							releaseModePallet[Index]			:= 1;
						ELSIF gSuperTrak.Par.Pallet[Index].IncrementOffset THEN
							releaseModePallet[Index]			:= 2;
						END_IF;

						// Do the same for motion parameters & release configS
						SuperTrakPalletParameters[Index].PalletConfig.Motion.Acceleration			:= gSuperTrak.Par.Pallet[Index].Config.Acceleration;
						SuperTrakPalletParameters[Index].PalletConfig.Motion.Velocity				:= gSuperTrak.Par.Pallet[Index].Config.Velocity;
						SuperTrakPalletParameters[Index].AdvancedReleaseConfig.DestinationTarget	:= gSuperTrak.Par.Pallet[Index].Config.DestinationTarget;
						SuperTrakPalletParameters[Index].AdvancedReleaseConfig.TargetOffset			:= gSuperTrak.Par.Pallet[Index].Config.TargetOffset;
						SuperTrakPalletParameters[Index].AdvancedReleaseConfig.IncrementalOffset	:= gSuperTrak.Par.Pallet[Index].Config.IncrementOffset;
						SuperTrakPalletParameters[Index].AdvancedReleaseConfig.Direction			:= gSuperTrak.Par.Pallet[Index].Config.Direction;

						StPalletState[Index]		:= 1;
					END_IF;
				1:	// Update motion parameters for the commanded movement
					StPallet_[Index].SetPalletMotionPar											:= TRUE;

					// Once the update is complete, move to the next state in the state machine
					IF StPallet_[Index].CommandDone THEN
						StPallet_[Index].SetPalletMotionPar										:= FALSE;
						StPalletState[Index]													:= 2;
					END_IF;
				2:
					// Update destination target and travel direction for the commanded movement
					StPallet_[Index].Update														:= TRUE;

					// Once the update is complete, move to the next state in the state machine
					IF StPallet_[Index].UpdateDone THEN
						StPallet_[Index].Update													:= FALSE;
						StPalletState[Index]													:= 3;
					END_IF;
				3:
					// Pass the ReleaseToTarget command onto the StTarget function block and execute
					CASE releaseModePallet[Index] OF
						0:		StPallet_[Index].ReleaseToTarget								:= TRUE;
						1:		StPallet_[Index].ReleaseToOffset								:= TRUE;
						2:		StPallet_[Index].IncrementOffset								:= TRUE;
					END_CASE;

					IF StPallet_[Index].CommandDone THEN
						StPallet_[Index].ReleaseToTarget										:= FALSE;
						StPallet_[Index].ReleaseToOffset										:= FALSE;
						StPallet_[Index].IncrementOffset										:= FALSE;
						StPalletState[Index]													:= 4;
					END_IF;

				4:	// Once the pallet is released, notify the main application w/ PalletReleased and reset the state machine
					gSuperTrak.Status.Pallet[Index].PalletReleased								:= TRUE;
					IF gSuperTrak.Par.Pallet[Index].ReleaseToTarget = FALSE AND gSuperTrak.Par.Pallet[Index].ReleaseToOffset = FALSE AND gSuperTrak.Par.Pallet[Index].IncrementOffset = FALSE THEN
						gSuperTrak.Status.Pallet[Index].PalletReleased							:= FALSE;
						StPalletState[Index]													:= 0;
					END_IF;
				5:
				6:
				7:
				8:
				9:
			END_CASE;
		END_FOR;

		// If the sections are not enabled, reset all commands
	ELSE
		// Loop thru all StTargetExt function blocks
		FOR Index := 0 TO (SIZEOF(StTargetExt_) / SIZEOF(StTargetExt_[0])) - 1 DO
			// Reset command
			StTargetExt_[Index].ReleaseToTarget   := FALSE;
		END_FOR;
	END_IF;

	(*************************************************************************************************)
	(*************************************************************************************************)
	(* ERROR RESET TO FUNCTION BLOCKS *)

	// Apply global Error Reset command to StControl FUB
	IF StControl_0.StatusID <> 0 THEN
		StControl_0.ErrorReset						:= gSuperTrak.Cmds.ErrorReset;
	ELSE
		StControl_0.ErrorReset						:= FALSE;
	END_IF;

	// Apply global Error Reset command to StTarget FUB
	FOR Index := 0 TO (SIZEOF(StTargetExt_) / SIZEOF(StTargetExt_[0])) -1 DO
		IF StTargetExt_[Index].StatusID <> 0 THEN
			StTargetExt_[Index].ErrorReset			:= gSuperTrak.Cmds.ErrorReset;
		ELSE
			StTargetExt_[Index].ErrorReset			:= FALSE;
		END_IF;
	END_FOR;

	// Apply global Error Reset command to StSection FUB
	FOR Index := 0 TO (SIZEOF(StSection_) / SIZEOF(StSection_[0])) - 1 DO
		IF StSection_[Index].StatusID <> 0 THEN
			StSection_[Index].ErrorReset			:= gSuperTrak.Cmds.ErrorReset;
		ELSE
			StSection_[Index].ErrorReset			:= FALSE;
		END_IF;
	END_FOR;

	// Apply global Error Reset command to StPallet FUB
	FOR Index := 0 TO (SIZEOF(StPallet_) / SIZEOF(StPallet_[0])) - 1 DO
		IF StPallet_[Index].StatusID <> 0 THEN
			StPallet_[Index].ErrorReset				:= gSuperTrak.Cmds.ErrorReset;
		ELSE
			StPallet_[Index].ErrorReset				:= FALSE;
		END_IF;
	END_FOR;

	(*************************************************************************************************)
	(*************************************************************************************************)
	(* FUNCTION BLOCK CALLS *)

	// Call StControl
	StControl_0();

	// Loop thru all StTargetExt function blocks
	FOR Index := 0 TO (SIZEOF(StSection_) / SIZEOF(StSection_[0])) - 1 DO
		// Call StSection
		StSection_[Index]();
	END_FOR;

	// Loop thru all StSection function blocks
	FOR Index := 0 TO (SIZEOF(StTargetExt_) / SIZEOF(StTargetExt_[0])) - 1 DO
		// Call StTargetExt
		StTargetExt_[Index]();
	END_FOR;

	// Loop thru all StPallet function blocks
	FOR Index := 0 TO (SIZEOF(StPallet_) / SIZEOF(StPallet_[0]))-1 DO
		// Call StPallet
		StPallet_[Index]();
	END_FOR;

	(*************************************************************************************************)
	(*************************************************************************************************)
	(* MAPPING OF STATUS VARIABLES *)

	SuperTrakGetPalletInfo(ADR(palletInfo),SIZEOF(palletInfo)/SIZEOF(palletInfo[0]),FALSE);

	//Actions to map status information into gSuperTrak structure

	ReadPNU;
//	WritePNU;
	GetStatus;

END_PROGRAM
```

#### Types.typ - Local data types
```iecst
(************************************************************************************************************************************)
(************************************************************************************************************************************)
(*Structures for SuperTrak control*)

TYPE
	SuperTrakCtrlType : 	STRUCT  (*Control structure for SuperTrak*)
		Command : SuperTrakCtrlCmdType; (*SuperTrak commands*)
		Parameter : SuperTrakCtrlParType; (*SuperTrak parameters*)
		Status : SuperTrakCtrlStatType; (*SuperTrak status*)
	END_STRUCT;
	SuperTrakCtrlCmdType : 	STRUCT  (*Command strucutre for SuperTrak*)
		EnableAllSections : BOOL; (*Command to enable all sections on the system*)
	END_STRUCT;
	SuperTrakCtrlParType : 	STRUCT  (*Parameter structure for SuperTrak*)
		Reserved : BOOL; (*Reserved for future development*)
	END_STRUCT;
	SuperTrakCtrlStatType : 	STRUCT  (*Status strucutre for SuperTrak*)
		AllSectionsEnabled : BOOL; (*Indicating if all sections on the system are enabled*)
	END_STRUCT;
	ReleaseStates_enum :
		(
		WAIT,
		SET_VEL,
		RELEASE,
		ERROR
		);
	WriteState_enum :
		(
		WS_WAIT,
		WS_SET_PARAMETERS,
		WS_WRITE,
		WS_APPLY,
		WS_ITERATE_SECTION,
		WS_DEBUG
		);
	ReadState_enum :
		(
		RS_WAIT := 0,
		RS_SET_PARAMETERS := 1,
		RS_READ := 2,
		RS_APPLY := 3,
		RS_ITERATE_SECTION := 4,
		RS_DEBUG := 5
		);
	Buffer_typ : 	STRUCT
		Entry : ARRAY[0..60]OF UINT;
	END_STRUCT;
END_TYPE
```

#### Variables.var - Local variables
```iecst
(************************************************************************************************************************************)
(************************************************************************************************************************************)
(************************************************************************************************************************************)
(************************************************************************************************************************************)
(*Function blocks*)
VAR
	StControl_0 : {REDUND_UNREPLICABLE} StControl; (*Function block to communicate to SuperTrak*)
	StSection_ : {REDUND_UNREPLICABLE} ARRAY[0..CONFIG_ST_MAX_SECTIONS] OF StSection; (*Function blocks to control SuperTrak sections*)
	StPallet_ : {REDUND_UNREPLICABLE} ARRAY[0..CONFIG_ST_MAX_PALLETS] OF StPallet;
	StTargetExt_ : {REDUND_UNREPLICABLE} ARRAY[0..CONFIG_ST_MAX_TARGETS] OF StTargetExt; (*Function blocks to control SuperTrak targets*)
END_VAR
(************************************************************************************************************************************)
(************************************************************************************************************************************)
(*Function block parameters*)
VAR
	SuperTrakControlParameters : {REDUND_UNREPLICABLE} StControlParType; (*Parameters for StControl*)
	SuperTrakPalletParameters : {REDUND_UNREPLICABLE} ARRAY[0..CONFIG_ST_MAX_PALLETS] OF StPalletParType;
	SuperTrakSectionParameters : {REDUND_UNREPLICABLE} ARRAY[0..CONFIG_ST_MAX_SECTIONS] OF StSectionParType; (*Parameters for StSection*)
	SuperTrakTargetParameters : {REDUND_UNREPLICABLE} ARRAY[0..CONFIG_ST_MAX_TARGETS] OF StTargetExtParType; (*Parameters for each StTargetExt*)
END_VAR
(************************************************************************************************************************************)
(************************************************************************************************************************************)
(*Other variables*)
VAR
	Index : {REDUND_UNREPLICABLE} USINT := 0; (*Index variable used in for loops*)
	StTargetState : ARRAY[0..CONFIG_ST_MAX_TARGETS] OF USINT;
	palletInfo : ARRAY[0..CONFIG_ST_MAX_PALLETS] OF SuperTrakPalletInfo_t;
	StPalletState : ARRAY[0..CONFIG_ST_MAX_PALLETS] OF USINT;
END_VAR
(************************************************************************************************************************************)
(************************************************************************************************************************************)
(*Read / Write variables*)
VAR
	StWritePnu_0 : StWritePnu;
	WritePnuPara : ARRAY[0..29] OF StWritePnuParType;
	ReadPnuPara : ARRAY[0..29] OF StReadPnuParType;
	StReadPnu_0 : StReadPnu;
END_VAR
VAR CONSTANT
	stSTAT_TARGET_PAR_VALUES : UINT := 1650;
	stSTAT_HARDWARE_SENSOR_VALUES : UINT := 1570;
END_VAR
VAR
	CurrentReadSection : USINT := 1;
	totalVelocity : REAL;
	averageVelocity : REAL;
	index : USINT;
END_VAR
VAR CONSTANT
	stNUM_WRITE_GROUPS : USINT := 1;
	stNUM_READ_GROUPS : USINT := 4;
END_VAR
VAR
	WriteDataBuffer : ARRAY[0..stNUM_WRITE_GROUPS] OF Buffer_typ;
	ReadDataBuffer : ARRAY[0..stNUM_READ_GROUPS] OF Buffer_typ;
END_VAR
VAR CONSTANT
	stSTAT_SECTION_TYPE : UINT := 1082;
	stSTAT_PALLET_DEST_TARGET : UINT := 1339;
	stSTAT_TARGET_POS_VALUES : UINT := 1651;
END_VAR
VAR
	nxt_adr : UDINT;
	releaseModeTarget : ARRAY[0..CONFIG_ST_MAX_TARGETS] OF USINT;
	releaseModePallet : ARRAY[0..CONFIG_ST_MAX_PALLETS] OF USINT;
	result : UINT;
	servChanResponseUINT : ARRAY[0..127] OF UINT;
	targetPositions : ARRAY[0..63] OF DINT;
	targetSections : ARRAY[0..127] OF UINT;
	sectionTemperatures : ARRAY[0..127] OF UINT;
	palletDestinations : ARRAY[0..127] OF UINT;
	sectionTypes : ARRAY[0..127] OF UINT;
	alphaEMA : REAL := 0.00004;
	palletVelocities : ARRAY[0..127] OF INT;
	palletAccelerations : ARRAY[0..127] OF UINT;
END_VAR
```

#### actReadWrite.st
```iecst
ACTION ReadPNU:

	// Read Target Section Values --------------------------------------------------------------------------------------------------------
	result		:= SuperTrakServChanRead( 0, stSTAT_TARGET_PAR_VALUES, 0, CONFIG_ST_MAX_TARGETS, ADR(servChanResponseUINT), SIZEOF(servChanResponseUINT));
	nxt_adr		:= memcpy(ADR(targetSections),ADR(servChanResponseUINT),SIZEOF(servChanResponseUINT));
	// Apply values
	FOR index := 0 TO CONFIG_ST_MAX_TARGETS DO
		gSuperTrak.Status.Target[index].Section			:= targetSections[index];
	END_FOR;

	// Read Target Position Values [initially um, converted to mm] -----------------------------------------------------------------------
	result		:= SuperTrakServChanRead( 0 , stSTAT_TARGET_POS_VALUES, 0, CONFIG_ST_MAX_TARGETS, ADR(servChanResponseUINT), SIZEOF(servChanResponseUINT));
	nxt_adr		:= memcpy(ADR(targetPositions),ADR(servChanResponseUINT),SIZEOF(servChanResponseUINT));
	// Apply values
	FOR index := 0 TO CONFIG_ST_MAX_TARGETS DO
		gSuperTrak.Status.Target[index].Position		:= DINT_TO_REAL(targetPositions[index]) / 1000.0;
	END_FOR;

	// Read Pallet Velocity Values -------------------------------------------------------------------------------------------------------
	result		:= SuperTrakServChanRead( 0, 1314, 0, CONFIG_ST_MAX_PALLETS, ADR(servChanResponseUINT), SIZEOF(servChanResponseUINT));
	nxt_adr		:= memcpy(ADR(palletVelocities),ADR(servChanResponseUINT),SIZEOF(servChanResponseUINT));
	// Apply values
	FOR index := 0 TO CONFIG_ST_MAX_PALLETS - 1 DO
		IF result = 0 THEN
			gSuperTrak.Status.Pallet[index+1].Velocity		:= UINT_TO_REAL(palletVelocities[index]);
		END_IF;
	END_FOR;

	// Read Pallet Acceleration Values ---------------------------------------------------------------------------------------------------
	result		:= SuperTrakServChanRead( 0, 1312, 0, CONFIG_ST_MAX_PALLETS, ADR(servChanResponseUINT), SIZEOF(servChanResponseUINT));
	nxt_adr		:= memcpy(ADR(palletAccelerations),ADR(servChanResponseUINT),SIZEOF(servChanResponseUINT));
	// Apply values
	FOR index := 0 TO CONFIG_ST_MAX_PALLETS DO
		IF result = 0 THEN

			gSuperTrak.Status.Pallet[index].Acceleration	:= palletAccelerations[index];

		END_IF;
	END_FOR;

	// Read Section Temperature Values ---------------------------------------------------------------------------------------------------
	result		:= SuperTrakServChanRead( CurrentReadSection, stSTAT_HARDWARE_SENSOR_VALUES, 0, 16, ADR(servChanResponseUINT), SIZEOF(servChanResponseUINT));
	nxt_adr		:= memcpy(ADR(sectionTemperatures),ADR(servChanResponseUINT),SIZEOF(servChanResponseUINT));
	// Apply values
	gSuperTrak.Status.Section[CurrentReadSection].Left.MotorTemp[1]			:= UINT_TO_REAL(sectionTemperatures[0]) / 100.0;
	gSuperTrak.Status.Section[CurrentReadSection].Left.MotorTemp[2]			:= UINT_TO_REAL(sectionTemperatures[1]) / 100.0;
	gSuperTrak.Status.Section[CurrentReadSection].Left.MotorTemp[3]			:= UINT_TO_REAL(sectionTemperatures[2]) / 100.0;
	gSuperTrak.Status.Section[CurrentReadSection].Left.MotorTemp[4]			:= UINT_TO_REAL(sectionTemperatures[3]) / 100.0;
	gSuperTrak.Status.Section[CurrentReadSection].Left.MotorTemp[5]			:= UINT_TO_REAL(sectionTemperatures[4]) / 100.0;
	gSuperTrak.Status.Section[CurrentReadSection].Left.ElectronicsTemp		:= UINT_TO_REAL(sectionTemperatures[5]) / 100.0;
	gSuperTrak.Status.Section[CurrentReadSection].Left.MotorVoltage			:= UINT_TO_REAL(sectionTemperatures[6]) / 100.0;

	gSuperTrak.Status.Section[CurrentReadSection].Right.MotorTemp[1]		:= UINT_TO_REAL(sectionTemperatures[0]) / 100.0;
	gSuperTrak.Status.Section[CurrentReadSection].Right.MotorTemp[2]		:= UINT_TO_REAL(sectionTemperatures[1]) / 100.0;
	gSuperTrak.Status.Section[CurrentReadSection].Right.MotorTemp[3]		:= UINT_TO_REAL(sectionTemperatures[2]) / 100.0;
	gSuperTrak.Status.Section[CurrentReadSection].Right.MotorTemp[4]		:= UINT_TO_REAL(sectionTemperatures[3]) / 100.0;
	gSuperTrak.Status.Section[CurrentReadSection].Right.MotorTemp[5]		:= UINT_TO_REAL(sectionTemperatures[4]) / 100.0;
	gSuperTrak.Status.Section[CurrentReadSection].Right.ElectronicsTemp		:= UINT_TO_REAL(sectionTemperatures[5]) / 100.0;
	gSuperTrak.Status.Section[CurrentReadSection].Right.MotorVoltage		:= UINT_TO_REAL(sectionTemperatures[6]) / 100.0;

	// Read Pallet Destination Targets ----------------------------------------------------------------------------------------------------
	result		:= SuperTrakServChanRead( 0, stSTAT_PALLET_DEST_TARGET, 0, CONFIG_ST_MAX_PALLETS, ADR(servChanResponseUINT), SIZEOF(servChanResponseUINT));
	nxt_adr		:= memcpy(ADR(palletDestinations),ADR(servChanResponseUINT),SIZEOF(servChanResponseUINT));
	// Apply values
	FOR index := 0 TO (CONFIG_ST_MAX_PALLETS - 1) DO
		gSuperTrak.Status.Pallet[index+1].DestinationTarget		:= palletDestinations[index];
	END_FOR;

	// Read Section Types ------------------------------------------------------------------------------------------------------------------
	result		:= SuperTrakServChanRead( CurrentReadSection, stSTAT_SECTION_TYPE, 0, 1, ADR(servChanResponseUINT), SIZEOF(servChanResponseUINT));
	nxt_adr		:= memcpy(ADR(sectionTypes),ADR(servChanResponseUINT),SIZEOF(servChanResponseUINT));
	// Apply values
	gSuperTrak.Status.Section[CurrentReadSection].IsCurveSection			:= UINT_TO_BOOL(sectionTypes[0]);

	// Index CurrentReadSection, used by some reads above
	CurrentReadSection				:= CurrentReadSection + 1;
	IF CurrentReadSection > CONFIG_ST_MAX_SECTIONS THEN
		CurrentReadSection	:= 1;
	END_IF;

END_ACTION

ACTION WritePNU:

	StWritePnu_0.Enable									:= StControl_0.Active;

	// Example write - PNU 1600 is for Region Options
	WritePnuPara[0].ValidDataSize						:= 4;
	WritePnuPara[0].ParameterNumber						:= 1600;
	WritePnuPara[0].ParameterValueCount					:= 2;
	WritePnuPara[0].SectionID							;	//	:= CurrentWriteSection;
	WritePnuPara[0].StartParameterIndex					:= 0;

	CASE WriteState OF

		WS_WAIT://-----------------------------------------------------------------------

			// Timer adds a small delay to manage system resource usage
			hwParameterWriteTimer.PT				:= t#1s;
			hwParameterWriteTimer.IN				:= TRUE;

			StWritePnu_0.Update						:= FALSE;
			StWritePnu_0.Write						:= FALSE;

			IF hwParameterWriteTimer.Q THEN
				hwParameterWriteTimer.IN			:= FALSE;
				WriteState							:= WS_APPLY;
			END_IF;

		WS_APPLY://-------------------------------------------------------------------------------

			IF enableRegionSample THEN
				WriteDataBuffer[0].Entry[0]			:= 3;
				WriteDataBuffer[0].Entry[1]			:= 3;
			ELSE
				WriteDataBuffer[0].Entry[0]			:= 2;
				WriteDataBuffer[0].Entry[1]			:= 2;
			END_IF;

			WriteState								:= WS_SET_PARAMETERS;

		WS_SET_PARAMETERS://-----------------------------------------------------------------------

			StWritePnu_0.Parameters					:= ADR(WritePnuPara[writeIndex]);
			StWritePnu_0.DataAddress				:= ADR(WriteDataBuffer[writeIndex].Entry);
			StWritePnu_0.DataSize					:= SIZEOF(WriteDataBuffer[writeIndex].Entry);

			StWritePnu_0.Update						:= TRUE;

			IF StWritePnu_0.UpdateDone THEN
				StWritePnu_0.Update					:= FALSE;
				WriteState							:= WS_WRITE;
			END_IF;

		WS_WRITE://-----------------------------------------------------------------------

			StWritePnu_0.Write						:= TRUE;

			IF StWritePnu_0.CommandDone THEN
				StWritePnu_0.Write					:= FALSE;
				WriteState							:= WS_ITERATE_SECTION;
			END_IF;

		WS_ITERATE_SECTION://-----------------------------------------------------------------------

			writeIndex								:= writeIndex + 1;
			WriteState								:= WS_APPLY;

			IF writeIndex = stNUM_WRITE_GROUPS THEN
				writeIndex							:= 0;
				CurrentWriteSection					:= CurrentWriteSection + 1;
				WriteState							:= WS_WAIT;
			END_IF;

			IF ( CurrentWriteSection < 1 ) OR ( CurrentWriteSection > CONFIG_ST_MAX_SECTIONS ) THEN
				CurrentWriteSection					:= 1;
			END_IF;

		WS_DEBUG://-----------------------------------------------------------------------

	END_CASE;

	hwParameterWriteTimer();
	StWritePnu_0();

END_ACTION
```

#### actGetStatus.st
```iecst
ACTION GetStatus:

	// This action maps all status bits from StControl, StPallet, and StTarget into the gSuperTrak global structure

	gSuperTrak.Status.System.Enabled   								:= StControl_0.SectionsEnabled;

	gSuperTrak.Status.System.FaultsActive							:= StControl_0.Info.SuperTrak.SystemFaultActive;
	gSuperTrak.Status.System.WarningActive							:= StControl_0.Info.SuperTrak.SystemWarningActive;

	// Would like to iterate through a FOR loop, but the bitwise structure of StControl prevents this.
	gSuperTrak.Status.System.Warnings[0]							:= StControl_0.Info.SuperTrak.SystemWarningBits.0;
	gSuperTrak.Status.System.Warnings[1]							:= StControl_0.Info.SuperTrak.SystemWarningBits.1;
	gSuperTrak.Status.System.Warnings[2]							:= StControl_0.Info.SuperTrak.SystemWarningBits.2;
	gSuperTrak.Status.System.Warnings[3]							:= StControl_0.Info.SuperTrak.SystemWarningBits.3;
	gSuperTrak.Status.System.Warnings[4]							:= StControl_0.Info.SuperTrak.SystemWarningBits.4;
	gSuperTrak.Status.System.Warnings[5]							:= StControl_0.Info.SuperTrak.SystemWarningBits.5;
	gSuperTrak.Status.System.Warnings[6]							:= StControl_0.Info.SuperTrak.SystemWarningBits.6;
	gSuperTrak.Status.System.Warnings[7]							:= StControl_0.Info.SuperTrak.SystemWarningBits.7;
	gSuperTrak.Status.System.Warnings[8]							:= StControl_0.Info.SuperTrak.SystemWarningBits.8;
	gSuperTrak.Status.System.Warnings[9]							:= StControl_0.Info.SuperTrak.SystemWarningBits.9;
	gSuperTrak.Status.System.Warnings[10]							:= StControl_0.Info.SuperTrak.SystemWarningBits.10;
	gSuperTrak.Status.System.Warnings[11]							:= StControl_0.Info.SuperTrak.SystemWarningBits.11;
	gSuperTrak.Status.System.Warnings[12]							:= StControl_0.Info.SuperTrak.SystemWarningBits.12;
	gSuperTrak.Status.System.Warnings[13]							:= StControl_0.Info.SuperTrak.SystemWarningBits.13;
	gSuperTrak.Status.System.Warnings[14]							:= StControl_0.Info.SuperTrak.SystemWarningBits.14;
	gSuperTrak.Status.System.Warnings[15]							:= StControl_0.Info.SuperTrak.SystemWarningBits.15;
	gSuperTrak.Status.System.Warnings[16]							:= StControl_0.Info.SuperTrak.SystemWarningBits.16;
	gSuperTrak.Status.System.Warnings[17]							:= StControl_0.Info.SuperTrak.SystemWarningBits.17;
	gSuperTrak.Status.System.Warnings[18]							:= StControl_0.Info.SuperTrak.SystemWarningBits.18;
	gSuperTrak.Status.System.Warnings[19]							:= StControl_0.Info.SuperTrak.SystemWarningBits.19;
	gSuperTrak.Status.System.Warnings[20]							:= StControl_0.Info.SuperTrak.SystemWarningBits.20;
	gSuperTrak.Status.System.Warnings[21]							:= StControl_0.Info.SuperTrak.SystemWarningBits.21;
	gSuperTrak.Status.System.Warnings[22]							:= StControl_0.Info.SuperTrak.SystemWarningBits.22;
	gSuperTrak.Status.System.Warnings[23]							:= StControl_0.Info.SuperTrak.SystemWarningBits.23;
	gSuperTrak.Status.System.Warnings[24]							:= StControl_0.Info.SuperTrak.SystemWarningBits.24;
	gSuperTrak.Status.System.Warnings[25]							:= StControl_0.Info.SuperTrak.SystemWarningBits.25;
	gSuperTrak.Status.System.Warnings[26]							:= StControl_0.Info.SuperTrak.SystemWarningBits.26;
	gSuperTrak.Status.System.Warnings[27]							:= StControl_0.Info.SuperTrak.SystemWarningBits.27;
	gSuperTrak.Status.System.Warnings[28]							:= StControl_0.Info.SuperTrak.SystemWarningBits.28;
	gSuperTrak.Status.System.Warnings[29]							:= StControl_0.Info.SuperTrak.SystemWarningBits.29;
	gSuperTrak.Status.System.Warnings[30]							:= StControl_0.Info.SuperTrak.SystemWarningBits.30;

	gSuperTrak.Status.System.Faults[0]								:= StControl_0.Info.SuperTrak.SystemFaultBits.0;
	gSuperTrak.Status.System.Faults[1]								:= StControl_0.Info.SuperTrak.SystemFaultBits.1;
	gSuperTrak.Status.System.Faults[2]								:= StControl_0.Info.SuperTrak.SystemFaultBits.2;
	gSuperTrak.Status.System.Faults[3]								:= StControl_0.Info.SuperTrak.SystemFaultBits.3;
	gSuperTrak.Status.System.Faults[4]								:= StControl_0.Info.SuperTrak.SystemFaultBits.4;
	gSuperTrak.Status.System.Faults[5]								:= StControl_0.Info.SuperTrak.SystemFaultBits.5;
	gSuperTrak.Status.System.Faults[6]								:= StControl_0.Info.SuperTrak.SystemFaultBits.6;
	gSuperTrak.Status.System.Faults[7]								:= StControl_0.Info.SuperTrak.SystemFaultBits.7;
	gSuperTrak.Status.System.Faults[8]								:= StControl_0.Info.SuperTrak.SystemFaultBits.8;
	gSuperTrak.Status.System.Faults[9]								:= StControl_0.Info.SuperTrak.SystemFaultBits.9;
	gSuperTrak.Status.System.Faults[10]								:= StControl_0.Info.SuperTrak.SystemFaultBits.10;
	gSuperTrak.Status.System.Faults[11]								:= StControl_0.Info.SuperTrak.SystemFaultBits.11;
	gSuperTrak.Status.System.Faults[12]								:= StControl_0.Info.SuperTrak.SystemFaultBits.12;
	gSuperTrak.Status.System.Faults[13]								:= StControl_0.Info.SuperTrak.SystemFaultBits.13;
	gSuperTrak.Status.System.Faults[14]								:= StControl_0.Info.SuperTrak.SystemFaultBits.14;
	gSuperTrak.Status.System.Faults[15]								:= StControl_0.Info.SuperTrak.SystemFaultBits.15;
	gSuperTrak.Status.System.Faults[16]								:= StControl_0.Info.SuperTrak.SystemFaultBits.16;
	gSuperTrak.Status.System.Faults[17]								:= StControl_0.Info.SuperTrak.SystemFaultBits.17;
	gSuperTrak.Status.System.Faults[18]								:= StControl_0.Info.SuperTrak.SystemFaultBits.18;
	gSuperTrak.Status.System.Faults[19]								:= StControl_0.Info.SuperTrak.SystemFaultBits.19;
	gSuperTrak.Status.System.Faults[20]								:= StControl_0.Info.SuperTrak.SystemFaultBits.20;
	gSuperTrak.Status.System.Faults[21]								:= StControl_0.Info.SuperTrak.SystemFaultBits.21;
	gSuperTrak.Status.System.Faults[22]								:= StControl_0.Info.SuperTrak.SystemFaultBits.22;
	gSuperTrak.Status.System.Faults[23]								:= StControl_0.Info.SuperTrak.SystemFaultBits.23;
	gSuperTrak.Status.System.Faults[24]								:= StControl_0.Info.SuperTrak.SystemFaultBits.24;
	gSuperTrak.Status.System.Faults[25]								:= StControl_0.Info.SuperTrak.SystemFaultBits.25;
	gSuperTrak.Status.System.Faults[26]								:= StControl_0.Info.SuperTrak.SystemFaultBits.26;
	gSuperTrak.Status.System.Faults[27]								:= StControl_0.Info.SuperTrak.SystemFaultBits.27;
	gSuperTrak.Status.System.Faults[28]								:= StControl_0.Info.SuperTrak.SystemFaultBits.28;
	gSuperTrak.Status.System.Faults[29]								:= StControl_0.Info.SuperTrak.SystemFaultBits.29;
	gSuperTrak.Status.System.Faults[30]								:= StControl_0.Info.SuperTrak.SystemFaultBits.30;

	// Start by assuming system is Ready. Code below conditionally resets
	gSuperTrak.Status.System.Ready									:= TRUE;

	// Start by assuming zero active sections. Code below conditionally resets
	gSuperTrak.Status.System.ActiveSections							:= 0;

	FOR Index := 0 TO SIZEOF(StSection_) / SIZEOF(StSection_[0]) - 1 DO

		// Then count sections with a Status other than zero
		IF StSection_[Index].Section <> 0 THEN
			gSuperTrak.Status.System.ActiveSections					:= gSuperTrak.Status.System.ActiveSections + 1;
		END_IF;

		// Verbose mapping of status bits to gSuperTrak structure
		gSuperTrak.Status.Section[Index].Diag.Enabled				:= StSection_[Index].SectionEnabled;
		gSuperTrak.Status.Section[Index].Diag.UnrecPallPresent		:= StSection_[Index].UnrecognizedPallets;
		gSuperTrak.Status.Section[Index].Diag.MotorPowerOn			:= StSection_[Index].MotorPowerOn;
		gSuperTrak.Status.Section[Index].Diag.PalletsRecovering		:= StSection_[Index].PalletsRecovering;
		gSuperTrak.Status.Section[Index].Diag.LocatingPallets		:= StSection_[Index].LocatingPallets;
		gSuperTrak.Status.Section[Index].Diag.DisabledExternally	:= StSection_[Index].DisabledExternally OR StSection_[Index].Info.SuperTrak.SectionFaultBits.28;

		gSuperTrak.Status.Section[Index].Diag.FaultActive			:= StSection_[Index].Info.SuperTrak.SectionFaultActive;
		gSuperTrak.Status.Section[Index].Diag.WarningActive			:= StSection_[Index].Info.SuperTrak.SectionWarningActive;

		gSuperTrak.Status.Section[Index].Diag.Faults[0]				:= StSection_[Index].Info.SuperTrak.SectionFaultBits.0;
		gSuperTrak.Status.Section[Index].Diag.Faults[1]				:= StSection_[Index].Info.SuperTrak.SectionFaultBits.1;
		gSuperTrak.Status.Section[Index].Diag.Faults[2]				:= StSection_[Index].Info.SuperTrak.SectionFaultBits.2;
		gSuperTrak.Status.Section[Index].Diag.Faults[3]				:= StSection_[Index].Info.SuperTrak.SectionFaultBits.3;
		gSuperTrak.Status.Section[Index].Diag.Faults[4]				:= StSection_[Index].Info.SuperTrak.SectionFaultBits.4;
		gSuperTrak.Status.Section[Index].Diag.Faults[5]				:= StSection_[Index].Info.SuperTrak.SectionFaultBits.5;
		gSuperTrak.Status.Section[Index].Diag.Faults[6]				:= StSection_[Index].Info.SuperTrak.SectionFaultBits.6;
		gSuperTrak.Status.Section[Index].Diag.Faults[7]				:= StSection_[Index].Info.SuperTrak.SectionFaultBits.7;
		gSuperTrak.Status.Section[Index].Diag.Faults[8]				:= StSection_[Index].Info.SuperTrak.SectionFaultBits.8;
		gSuperTrak.Status.Section[Index].Diag.Faults[9]				:= StSection_[Index].Info.SuperTrak.SectionFaultBits.9;
		gSuperTrak.Status.Section[Index].Diag.Faults[10]			:= StSection_[Index].Info.SuperTrak.SectionFaultBits.10;
		gSuperTrak.Status.Section[Index].Diag.Faults[11]			:= StSection_[Index].Info.SuperTrak.SectionFaultBits.11;
		gSuperTrak.Status.Section[Index].Diag.Faults[12]			:= StSection_[Index].Info.SuperTrak.SectionFaultBits.12;
		gSuperTrak.Status.Section[Index].Diag.Faults[13]			:= StSection_[Index].Info.SuperTrak.SectionFaultBits.13;
		gSuperTrak.Status.Section[Index].Diag.Faults[14]			:= StSection_[Index].Info.SuperTrak.SectionFaultBits.14;
		gSuperTrak.Status.Section[Index].Diag.Faults[15]			:= StSection_[Index].Info.SuperTrak.SectionFaultBits.15;
		gSuperTrak.Status.Section[Index].Diag.Faults[16]			:= StSection_[Index].Info.SuperTrak.SectionFaultBits.16;
		gSuperTrak.Status.Section[Index].Diag.Faults[17]			:= StSection_[Index].Info.SuperTrak.SectionFaultBits.17;
		gSuperTrak.Status.Section[Index].Diag.Faults[18]			:= StSection_[Index].Info.SuperTrak.SectionFaultBits.18;
		gSuperTrak.Status.Section[Index].Diag.Faults[19]			:= StSection_[Index].Info.SuperTrak.SectionFaultBits.19;
		gSuperTrak.Status.Section[Index].Diag.Faults[20]			:= StSection_[Index].Info.SuperTrak.SectionFaultBits.20;
		gSuperTrak.Status.Section[Index].Diag.Faults[21]			:= StSection_[Index].Info.SuperTrak.SectionFaultBits.21;
		gSuperTrak.Status.Section[Index].Diag.Faults[22]			:= StSection_[Index].Info.SuperTrak.SectionFaultBits.22;
		gSuperTrak.Status.Section[Index].Diag.Faults[23]			:= StSection_[Index].Info.SuperTrak.SectionFaultBits.23;
		gSuperTrak.Status.Section[Index].Diag.Faults[24]			:= StSection_[Index].Info.SuperTrak.SectionFaultBits.24;
		gSuperTrak.Status.Section[Index].Diag.Faults[25]			:= StSection_[Index].Info.SuperTrak.SectionFaultBits.25;
		gSuperTrak.Status.Section[Index].Diag.Faults[26]			:= StSection_[Index].Info.SuperTrak.SectionFaultBits.26;
		gSuperTrak.Status.Section[Index].Diag.Faults[27]			:= StSection_[Index].Info.SuperTrak.SectionFaultBits.27;
		gSuperTrak.Status.Section[Index].Diag.Faults[28]			:= StSection_[Index].Info.SuperTrak.SectionFaultBits.28;
		gSuperTrak.Status.Section[Index].Diag.Faults[29]			:= StSection_[Index].Info.SuperTrak.SectionFaultBits.29;
		gSuperTrak.Status.Section[Index].Diag.Faults[30]			:= StSection_[Index].Info.SuperTrak.SectionFaultBits.30;
		gSuperTrak.Status.Section[Index].Diag.Faults[31]			:= StSection_[Index].Info.SuperTrak.SectionFaultBits.31;

		gSuperTrak.Status.Section[Index].Diag.Warnings[0]			:= StSection_[Index].Info.SuperTrak.SectionWarningBits.0;
		gSuperTrak.Status.Section[Index].Diag.Warnings[1]			:= StSection_[Index].Info.SuperTrak.SectionWarningBits.1;
		gSuperTrak.Status.Section[Index].Diag.Warnings[2]			:= StSection_[Index].Info.SuperTrak.SectionWarningBits.2;
		gSuperTrak.Status.Section[Index].Diag.Warnings[3]			:= StSection_[Index].Info.SuperTrak.SectionWarningBits.3;
		gSuperTrak.Status.Section[Index].Diag.Warnings[4]			:= StSection_[Index].Info.SuperTrak.SectionWarningBits.4;
		gSuperTrak.Status.Section[Index].Diag.Warnings[5]			:= StSection_[Index].Info.SuperTrak.SectionWarningBits.5;
		gSuperTrak.Status.Section[Index].Diag.Warnings[6]			:= StSection_[Index].Info.SuperTrak.SectionWarningBits.6;
		gSuperTrak.Status.Section[Index].Diag.Warnings[7]			:= StSection_[Index].Info.SuperTrak.SectionWarningBits.7;
		gSuperTrak.Status.Section[Index].Diag.Warnings[8]			:= StSection_[Index].Info.SuperTrak.SectionWarningBits.8;
		gSuperTrak.Status.Section[Index].Diag.Warnings[9]			:= StSection_[Index].Info.SuperTrak.SectionWarningBits.9;
		gSuperTrak.Status.Section[Index].Diag.Warnings[10]			:= StSection_[Index].Info.SuperTrak.SectionWarningBits.10;
		gSuperTrak.Status.Section[Index].Diag.Warnings[11]			:= StSection_[Index].Info.SuperTrak.SectionWarningBits.11;
		gSuperTrak.Status.Section[Index].Diag.Warnings[12]			:= StSection_[Index].Info.SuperTrak.SectionWarningBits.12;
		gSuperTrak.Status.Section[Index].Diag.Warnings[13]			:= StSection_[Index].Info.SuperTrak.SectionWarningBits.13;
		gSuperTrak.Status.Section[Index].Diag.Warnings[14]			:= StSection_[Index].Info.SuperTrak.SectionWarningBits.14;
		gSuperTrak.Status.Section[Index].Diag.Warnings[15]			:= StSection_[Index].Info.SuperTrak.SectionWarningBits.15;
		gSuperTrak.Status.Section[Index].Diag.Warnings[16]			:= StSection_[Index].Info.SuperTrak.SectionWarningBits.16;
		gSuperTrak.Status.Section[Index].Diag.Warnings[17]			:= StSection_[Index].Info.SuperTrak.SectionWarningBits.17;
		gSuperTrak.Status.Section[Index].Diag.Warnings[18]			:= StSection_[Index].Info.SuperTrak.SectionWarningBits.18;
		gSuperTrak.Status.Section[Index].Diag.Warnings[19]			:= StSection_[Index].Info.SuperTrak.SectionWarningBits.19;
		gSuperTrak.Status.Section[Index].Diag.Warnings[20]			:= StSection_[Index].Info.SuperTrak.SectionWarningBits.20;
		gSuperTrak.Status.Section[Index].Diag.Warnings[21]			:= StSection_[Index].Info.SuperTrak.SectionWarningBits.21;
		gSuperTrak.Status.Section[Index].Diag.Warnings[22]			:= StSection_[Index].Info.SuperTrak.SectionWarningBits.22;
		gSuperTrak.Status.Section[Index].Diag.Warnings[23]			:= StSection_[Index].Info.SuperTrak.SectionWarningBits.23;
		gSuperTrak.Status.Section[Index].Diag.Warnings[24]			:= StSection_[Index].Info.SuperTrak.SectionWarningBits.24;
		gSuperTrak.Status.Section[Index].Diag.Warnings[25]			:= StSection_[Index].Info.SuperTrak.SectionWarningBits.25;
		gSuperTrak.Status.Section[Index].Diag.Warnings[26]			:= StSection_[Index].Info.SuperTrak.SectionWarningBits.26;
		gSuperTrak.Status.Section[Index].Diag.Warnings[27]			:= StSection_[Index].Info.SuperTrak.SectionWarningBits.27;
		gSuperTrak.Status.Section[Index].Diag.Warnings[28]			:= StSection_[Index].Info.SuperTrak.SectionWarningBits.28;
		gSuperTrak.Status.Section[Index].Diag.Warnings[29]			:= StSection_[Index].Info.SuperTrak.SectionWarningBits.29;
		gSuperTrak.Status.Section[Index].Diag.Warnings[30]			:= StSection_[Index].Info.SuperTrak.SectionWarningBits.30;
		gSuperTrak.Status.Section[Index].Diag.Warnings[31]			:= StSection_[Index].Info.SuperTrak.SectionWarningBits.31;

		// Status Ready bit. Pallets should be recovered and all sections
		IF Index <> 0 THEN
			IF (gSuperTrak.Status.Section[Index].Diag.Enabled = FALSE) OR (gSuperTrak.Status.Section[Index].Diag.PalletsRecovering = TRUE) OR (gSuperTrak.Status.Section[Index].Diag.LocatingPallets = TRUE) THEN
				gSuperTrak.Status.System.Ready						:= FALSE;
			END_IF;
		END_IF;
	END_FOR;

	// Map target status bits to gSuperTrak
	FOR Index := 0 TO SIZEOF(StTargetExt_) / SIZEOF(StTargetExt_[0])-1 DO
		gSuperTrak.Status.Target[Index].PalletId					:= StTargetExt_[Index].PalletID;
		gSuperTrak.Status.Target[Index].PalletPresent				:= StTargetExt_[Index].PalletPresent;
		gSuperTrak.Status.Target[Index].PalletPreArrival			:= StTargetExt_[Index].PalletPreArrival;
		gSuperTrak.Status.Target[Index].PalletHovering				:= StTargetExt_[Index].PalletOverTarget;
	END_FOR;

	// Start by assuming active pallets zero
	gSuperTrak.Status.System.ActivePallets							:= 0;

	// Calculation for instantaneous throughput of shuttles [shuttles/s]
	// AverageShuttleVelocity [m/s] * ShuttleCount [] / TotalTrackLength [m]
	// Start AverageShuttleVelocity calculation by assuming totalVelocity is zero
	totalVelocity													:= 0;

	FOR Index := 0 TO (SIZEOF(StPallet_) / SIZEOF(StPallet_[0]))-2 DO

		// Map pallet status bits to gSuperTrak
		gSuperTrak.Status.Pallet[Index+1].Position					:= DINT_TO_REAL(palletInfo[Index].position) / 1000.0;
		gSuperTrak.Status.Pallet[Index+1].Section					:= palletInfo[Index].section;
		gSuperTrak.Status.Pallet[Index+1].PalletAllocated			:= (palletInfo[Index].status <> 0);

		// For active pallets, sum all velocities
		IF gSuperTrak.Status.Pallet[Index+1].PalletAllocated THEN
			gSuperTrak.Status.System.ActivePallets					:= gSuperTrak.Status.System.ActivePallets + 1;
			totalVelocity											:= totalVelocity + gSuperTrak.Status.Pallet[Index+1].Velocity / 1000.0;
		END_IF;

	END_FOR;

	// Protect div0
	IF gSuperTrak.Status.System.ActiveSections <> 0 AND gSuperTrak.Status.System.ActivePallets <> 0 THEN
		// Divide by shuttle count to calculate AverageShuttleVelocity
		averageVelocity											:= totalVelocity / USINT_TO_REAL(gSuperTrak.Status.System.ActivePallets);
		// Calculate system throughput [shuttles/min]
		gSuperTrak.Status.System.Throughput						:= USINT_TO_REAL(gSuperTrak.Status.System.ActivePallets) * averageVelocity * 60.0 / USINT_TO_REAL(gSuperTrak.Status.System.ActiveSections);
		// Calculate Exponential weighted moving average. Weighting factor 'alphaEMA' can be modified to make this measurement more or less responsive
		gSuperTrak.Status.System.EMA_Throughput					:= ( alphaEMA * gSuperTrak.Status.System.Throughput ) + (( 1.0 - alphaEMA ) * gSuperTrak.Status.System.EMA_Throughput );
	ELSE
		gSuperTrak.Status.System.Throughput						:= 0.0;
		gSuperTrak.Status.System.EMA_Throughput					:= 0.0;
	END_IF;

END_ACTION
```

### Program Logical/Source/ST_Core/ST_Visu (IEC)

#### Cyclic.st - Cyclic code
```iecst
(*********************************************************************************
 * Copyright Bernecker + Rainer 2015
 * Copyright ATS Automation Tooling Systems, Inc. 2017-2018
 * All rights reserved.
 * -------------------------------------------------------------------------------
 * This task calculates the actual pallet positions in the room based on the
 * section number and the position of the pallet in the section.
 * It is also hiding unused sections and/or pallets.
 * This data is then provided to B&R Scene Viewer.
 *********************************************************************************)

PROGRAM _INIT

	// Data for JavaScript SuperTrak Widget:

	FOR index := 1 TO CONFIG_ST_MAX_PALLETS DO
		//		{"value":7,"text":"Pallet 7"}
		dataProviderPallet[index]		:= '{"value":';
		strIndex		:= USINT_TO_STRING(index);
		nxt_adr			:= strcat(ADR(dataProviderPallet[index]),ADR(strIndex));
		nxt_adr			:= strcat(ADR(dataProviderPallet[index]),ADR(',"text":"Pallet '));
		nxt_adr			:= strcat(ADR(dataProviderPallet[index]),ADR(strIndex));
		nxt_adr			:= strcat(ADR(dataProviderPallet[index]),ADR('"}'));
	END_FOR;

	FOR index := 1 TO CONFIG_ST_MAX_TARGETS DO
		//		{"value":7,"text":"Target 7"}
		dataProviderTarget[index]		:= '{"value":';
		strIndex		:= USINT_TO_STRING(index);
		nxt_adr			:= strcat(ADR(dataProviderTarget[index]),ADR(strIndex));
		nxt_adr			:= strcat(ADR(dataProviderTarget[index]),ADR(',"text":"Target '));
		nxt_adr			:= strcat(ADR(dataProviderTarget[index]),ADR(strIndex));
		nxt_adr			:= strcat(ADR(dataProviderTarget[index]),ADR('"}'));
	END_FOR;

	FOR index := 1 TO CONFIG_ST_MAX_SECTIONS DO
		//		{"value":7,"text":"Section 7"}
		dataProviderSection[index]		:= '{"value":';
		strIndex		:= USINT_TO_STRING(index);
		nxt_adr			:= strcat(ADR(dataProviderSection[index]),ADR(strIndex));
		nxt_adr			:= strcat(ADR(dataProviderSection[index]),ADR(',"text":"Section '));
		nxt_adr			:= strcat(ADR(dataProviderSection[index]),ADR(strIndex));
		nxt_adr			:= strcat(ADR(dataProviderSection[index]),ADR('"}'));
	END_FOR;

	visuStep := 0;

END_PROGRAM

PROGRAM _CYCLIC

	CASE visuStep OF
		visuSTEP_INITIALIZE:
			visuStep := visuSTEP_GET_SECTION_COUNT;

		visuSTEP_GET_SECTION_COUNT:
			// read parameter 1080: section count
			result := SuperTrakServChanRead(0, 1080, 0, 1, ADR(sectionCount), SIZEOF(sectionCount));

			IF (result = scERR_SUCCESS) AND (sectionCount > 0) THEN
				visuStep := visuSTEP_GET_SECTION_ADDRS;
			ELSE
				visuStep := visuSTEP_ERROR;
			END_IF;

		visuSTEP_GET_SECTION_ADDRS:
			// read parameter 1081: section user address
			result := SuperTrakServChanRead(0, 1081, 0, sectionCount, ADR(servChanResponseUINT), SIZEOF(servChanResponseUINT));

			IF (result = scERR_SUCCESS) THEN
				FOR i := 0 TO sectionCount - 1 DO
					Section[i].userAddress := servChanResponseUINT[i];

					IF (Section[i].userAddress > 0) AND (Section[i].userAddress < 99) THEN
						sectionLookup[ Section[i].userAddress ] := i;
					END_IF;
				END_FOR;

				visuStep := visuSTEP_GET_SECTION_TYPES;
				i := 0;
			ELSE
				visuStep := visuSTEP_ERROR;
			END_IF;

		visuSTEP_GET_SECTION_TYPES:
			// read parameter 1082: section type
			result := SuperTrakServChanRead(UINT_TO_USINT(Section[i].userAddress), 1082, 0, 1, ADR(Section[i].sectionType), SIZEOF(UINT));

			IF (result = scERR_SUCCESS) THEN
				i := i + 1;

				IF (i >= sectionCount) THEN
					visuStep := visuSTEP_SETUP_SECTIONS;
				END_IF;
			ELSE
				visuStep := visuSTEP_ERROR;
			END_IF;

		visuSTEP_SETUP_SECTIONS:
			// Assign visualization models to sections.
			// Mostly assume that the layout is sensible.
			side := 0;
			sideLength[0] := 0;
			sideLength[1] := 0;
			position := 0;
			modelIndex := 0;

			FOR i := 0 TO sectionCount - 1 DO
				Section[i].side := -1;
				Section[i].modelIndex := -1;

				IF (Section[i].sectionType = SECTION_TYPE_1M) OR (Section[i].sectionType = SECTION_TYPE_1M_LP) THEN
					// Straight section models are indexed 0-31 (front) and 32-63 (back).
					IF (side < 2)
						AND (modelIndex >= (side * 32))
						AND (modelIndex < ((side + 1) * 32)) THEN

						Section[i].side := side;
						sideLength[side] := sideLength[side] + 1;

						Data.StraightSectionVisible[modelIndex] := TRUE;
						Section[i].modelIndex := modelIndex;
						modelIndex := modelIndex + 1;

						Section[i].positionX := position;

						IF (side = 0) THEN
							position := position + 1000;
						ELSE
							position := position - 1000;
						END_IF;
					END_IF;

				ELSIF (Section[i].sectionType = SECTION_TYPE_N180) OR (Section[i].sectionType = SECTION_TYPE_W180L) THEN
					// Advance to next side when a curve follows straights,
					// or when a curve already exists on the current side.
					IF (side < 2) AND ((sideLength[side] > 0) OR (curveHSection[side] >= 0)) THEN
						side := side + 1;

						IF (side = 1) THEN
							modelIndex := 64 - sideLength[0];
							Data.CurvePositionX := position;
						END_IF;
					END_IF;

					IF (side = 1) THEN
						curveSide := 1;
					ELSE
						curveSide := 0;
					END_IF;

					IF (curveHSection[curveSide] < 0) THEN
						Section[i].side := curveSide;
						curveHSection[curveSide] := i;

						IF (Section[i].sectionType = SECTION_TYPE_N180) THEN
							Data.N180SectionVisible[curveSide] := TRUE;
						ELSE
							Data.W180SectionVisible[curveSide] := TRUE;
						END_IF;

						curveType := Section[i].sectionType;
					END_IF;

				ELSIF (Section[i].sectionType = SECTION_TYPE_W180R) THEN
					IF (side = 1) THEN
						curveSide := 1;
					ELSE
						curveSide := 0;
					END_IF;

					Section[i].side := curveSide;

				ELSE
					// unhandled section type

				END_IF;
			END_FOR;

			IF (curveType = SECTION_TYPE_N180) THEN
				Data.StraightSectionPositionY := 0;
				straightPalletPositionY[0] := -236;
				straightPalletPositionY[1] := 236;
			ELSE	// W180
				Data.StraightSectionPositionY := 365.5;
				straightPalletPositionY[0] := -236;
				straightPalletPositionY[1] := 600.5;
			END_IF;

			visuStep := visuSTEP_RUN;

		visuSTEP_RUN:
			// get actual pallet positions
			SuperTrakGetPalletInfo(ADR(Pallet), 128, FALSE);

			FOR i := 0 TO 127 DO
				IF (Pallet[i].section >= 1) AND (Pallet[i].section <= 99) THEN
					h := sectionLookup[ Pallet[i].section ];
				ELSE
					h := -1;
				END_IF;

				IF (h >= 0) THEN
					// display this pallet
					Data.Pallet[i].Visible := TRUE;
					position := DINT_TO_REAL(Pallet[i].position) / 1000;

					IF (Section[h].sectionType = SECTION_TYPE_1M) OR (Section[h].sectionType = SECTION_TYPE_1M_LP) THEN
						IF (Section[h].side = 0) THEN
							Data.Pallet[i].X := Section[h].positionX + position;
							Data.Pallet[i].Y := straightPalletPositionY[0];
							Data.Pallet[i].RZ := 0;
						ELSE
							Data.Pallet[i].X := Section[h].positionX - position;
							Data.Pallet[i].Y := straightPalletPositionY[1];
							Data.Pallet[i].RZ := 180;
						END_IF;

					ELSIF (Section[h].sectionType = SECTION_TYPE_N180) THEN
						// approximate the shape of the curve
						IF (position <= 15) THEN
							Data.Pallet[i].X := position;
							Data.Pallet[i].Y := -236;
							Data.Pallet[i].RZ := 0;
						ELSIF (position < 1015) THEN
							angle := brmPI * (position - 15) / 1000;
							Data.Pallet[i].X := 15 + (355 * SIN(angle)) - (15 * SIN(angle * 3));
							Data.Pallet[i].Y := (-257 * COS(angle)) + (21 * COS(angle * 3));
							Data.Pallet[i].RZ := 90 - 90 * COS(angle);
						ELSE
							Data.Pallet[i].X := 1030 - position;
							Data.Pallet[i].Y := 236;
							Data.Pallet[i].RZ := 180;
						END_IF;

						IF (Section[h].side = 0) THEN
							Data.Pallet[i].X := -Data.Pallet[i].X;
							Data.Pallet[i].Y := -Data.Pallet[i].Y;
							Data.Pallet[i].RZ := Data.Pallet[i].RZ - 180;
						ELSE
							Data.Pallet[i].X := Data.Pallet[i].X + Data.CurvePositionX;
						END_IF;

					ELSIF (Section[h].sectionType = SECTION_TYPE_W180L) THEN
						IF (position > 100) THEN
							angle := (position - 100) / W180_RADIUS * 180 / brmPI;
							position := 100;
						ELSE
							angle := 0;
						END_IF;

						IF (Section[h].side = 0) THEN
							Data.Pallet[i].X := -position - W180_RADIUS * SIN(angle * brmPI / 180);
							Data.Pallet[i].Y := 181.75 + W180_RADIUS * COS(angle * brmPI / 180);
							angle := angle + 180;
						ELSE
							Data.Pallet[i].X := position + Data.CurvePositionX + W180_RADIUS * SIN(angle * brmPI / 180);
							Data.Pallet[i].Y := 181.75 - W180_RADIUS * COS(angle * brmPI / 180);
						END_IF;

						Data.Pallet[i].RZ := angle;

					ELSIF (Section[h].sectionType = SECTION_TYPE_W180R) THEN
						IF (position > 650) THEN
							angle := 180;
							position := 750 - position;
						ELSE
							angle := (position / W180_RADIUS * 180 / brmPI) + 90;
							position := 100;
						END_IF;

						IF (Section[h].side = 0) THEN
							angle := angle + 180;
							Data.Pallet[i].X := -position - W180_RADIUS * ABS(SIN(angle * brmPI / 180));
							Data.Pallet[i].Y := 181.75 - W180_RADIUS * ABS(COS(angle * brmPI / 180));
						ELSE
							Data.Pallet[i].X := position + Data.CurvePositionX + W180_RADIUS * ABS(SIN(angle * brmPI / 180));
							Data.Pallet[i].Y := 181.75 + W180_RADIUS * ABS(COS(angle * brmPI / 180));
						END_IF;

						Data.Pallet[i].RZ := angle;

					END_IF;

				ELSE
					// hide this pallet
					Data.Pallet[i].Visible := FALSE;
					Data.Pallet[i].X := 0;
					Data.Pallet[i].Y := 0;
					Data.Pallet[i].RZ := 0;

				END_IF;
			END_FOR;

		ELSE
			// error or unhandled state; do nothing

	END_CASE;

	SuperTrakPaperWidget;

END_PROGRAM
```

#### Types.typ - Local data types
```iecst
TYPE
	RoboVisuPallet_t : 	STRUCT
		Visible : BOOL; (*byte 0*)
		reserved_1 : USINT; (*byte 1*)
		Text : STRING[5]; (*Text / bytes 2-7*) (*STRING[n] = char[n + 1] = n characters plus terminator*)
		X : REAL; (*Position.X / bytes 8-11*)
		Y : REAL; (*Position.Y / bytes 12-15*)
		RZ : REAL; (*Orientation.RotZ / bytes 16-19*)
	END_STRUCT;
	RoboVisuData_t : 	STRUCT
		StraightSectionVisible : ARRAY[0..63]OF BOOL; (*bytes 0-63*)
		N180SectionVisible : ARRAY[0..1]OF BOOL; (*bytes 64-65*)
		W180SectionVisible : ARRAY[0..1]OF BOOL; (*bytes 66-67*)
		StraightSectionPositionY : REAL; (*bytes 68-71*)
		CurvePositionX : REAL; (*bytes 72-75*)
		reserved_76 : REAL; (*bytes 76-79*)
		reserved_80 : ARRAY[0..47]OF USINT; (*bytes 80-127*)
		reserved_128 : ARRAY[0..383]OF USINT; (*bytes 128-511*)
		Pallet : ARRAY[0..127]OF RoboVisuPallet_t; (*bytes 512-3071*)
	END_STRUCT;
	SectionInfo_t : 	STRUCT
		userAddress : UINT;
		sectionType : UINT;
		side : INT;
		modelIndex : INT;
		positionX : REAL;
	END_STRUCT;
	WidgetData_t : 	STRUCT
		SectionCount : USINT;
		ShuttleCount : USINT;
		ShuttlePos : ARRAY[0..CONFIG_ST_MAX_PALLETS]OF REAL;
		TargetPos : ARRAY[0..CONFIG_ST_MAX_TARGETS]OF REAL;
		TargetCount : USINT;
	END_STRUCT;
	ItemCollection_t : 	STRUCT
		first : STRING[50] := '{"value":1,"text":"Select 1"}';
		second : STRING[50] := '{"value":2,"text":"Select 2"}';
		third : STRING[50] := '{"value":3,"text":"Select 3"}';
	END_STRUCT;
END_TYPE
```

#### Variables.var - Local variables
```iecst
(*Visualization program states*)
VAR
	targetStatusIndex : USINT;
	palletStatusIndex : USINT;
	sectionStatusIndex : USINT;
	pPalletStatusRef : REFERENCE TO SysPalletStatus_typ;
	pSectionStatusRef : REFERENCE TO SysSectionStatus_typ;
	pTargetStatusRef : REFERENCE TO SysTargetStatus_typ;
END_VAR
VAR CONSTANT
	visuSTEP_INITIALIZE : USINT := 0;
	visuSTEP_GET_SECTION_COUNT : USINT := 1;
	visuSTEP_GET_SECTION_ADDRS : USINT := 2;
	visuSTEP_GET_SECTION_TYPES : USINT := 3;
	visuSTEP_SETUP_SECTIONS : USINT := 10;
	visuSTEP_RUN : USINT := 42;
	visuSTEP_ERROR : USINT := 99;
END_VAR
(*SuperTrak section types*)
VAR CONSTANT
	SECTION_TYPE_1M : UINT := 0;
	SECTION_TYPE_N180 : UINT := 1;
	SECTION_TYPE_1M_LP : UINT := 2;
	SECTION_TYPE_W180L : UINT := 3;
	SECTION_TYPE_W180R : UINT := 4;
END_VAR
(*Miscellaneous constants*)
VAR CONSTANT
	W180_RADIUS : REAL := 418.75;
END_VAR
(*Miscellaneous variables*)
VAR
	angle : REAL := 0.0;
	h : INT := 0;
	i : UINT := 0;
	position : REAL := 0.0;
	result : UINT := 0;
	index : USINT;
	visuStep : USINT := 0;
END_VAR
(*Visualization variables*)
VAR
	Data : RoboVisuData_t := (0); (*exported to Robotic Visualization*)
	sectionCount : UINT := 0;
	Section : ARRAY[0..63] OF SectionInfo_t; (*index = hSection*)
	Pallet : ARRAY[0..127] OF SuperTrakPalletInfo_t := [128(0)];
	sectionLookup : ARRAY[0..99] OF INT := [100(-1)]; (*index = user address, value = hSection*)
	straightPalletPositionY : ARRAY[0..1] OF REAL := [2(0.0)];
END_VAR
(*Setup variables*)
VAR
	curveHSection : ARRAY[0..1] OF INT := [2(-1)];
	curveSide : INT := 0;
	curveType : UINT := 0;
	modelIndex : INT := 0;
	side : INT := 0;
	sideLength : ARRAY[0..1] OF UINT := [2(0)];
END_VAR
(*SuperTrak service channel*)
VAR
	servChanResponseUINT : {REDUND_UNREPLICABLE} ARRAY[0..63] OF UINT;
	WidgetData : WidgetData_t;
	nxt_adr : UDINT;
	dataProviderSection : ARRAY[0..CONFIG_ST_MAX_SECTIONS] OF STRING[80];
	dataProviderTarget : ARRAY[0..CONFIG_ST_MAX_TARGETS] OF STRING[80];
	dataProviderPallet : ARRAY[0..CONFIG_ST_MAX_PALLETS] OF STRING[80];
	strIndex : STRING[50];
END_VAR
```
